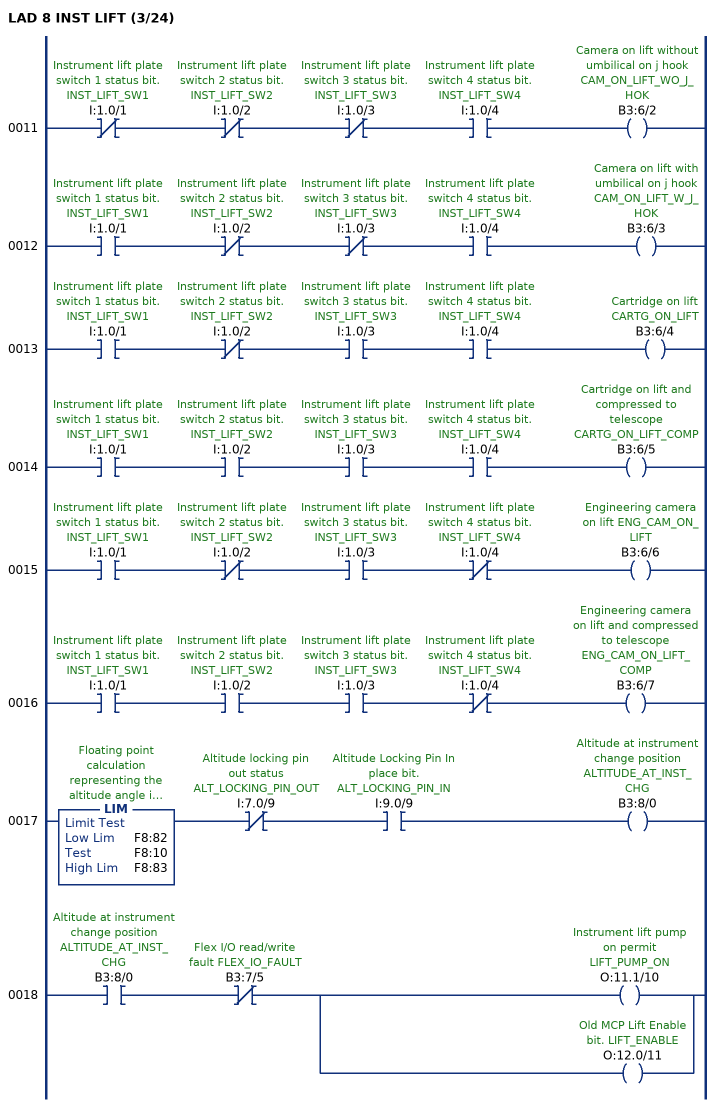
% Rung: 11 %
SOR XIO I:1.0/1 XIO I:1.0/2 XIO I:1.0/3 XIC I:1.0/4 OTE B3:6/2 EOR
%   I:1.0/1  INST_LIFT_SW1  "Instrument lift plate switch 1 status bit." %
%   I:1.0/2  INST_LIFT_SW2  "Instrument lift plate switch 2 status bit." %
%   I:1.0/3  INST_LIFT_SW3  "Instrument lift plate switch 3 status bit." %
%   I:1.0/4  INST_LIFT_SW4  "Instrument lift plate switch 4 status bit." %
%   B3:6/2  CAM_ON_LIFT_WO_J_HOK  "Camera on lift without umbilical on j hook" %
% Rung: 12 %
SOR XIC I:1.0/1 XIO I:1.0/2 XIO I:1.0/3 XIC I:1.0/4 OTE B3:6/3 EOR
%   I:1.0/1  INST_LIFT_SW1  "Instrument lift plate switch 1 status bit." %
%   I:1.0/2  INST_LIFT_SW2  "Instrument lift plate switch 2 status bit." %
%   I:1.0/3  INST_LIFT_SW3  "Instrument lift plate switch 3 status bit." %
%   I:1.0/4  INST_LIFT_SW4  "Instrument lift plate switch 4 status bit." %
%   B3:6/3  CAM_ON_LIFT_W_J_HOK  "Camera on lift with umbilical on j hook" %
% Rung: 13 %
SOR XIC I:1.0/1 XIO I:1.0/2 XIC I:1.0/3 XIC I:1.0/4 OTE B3:6/4 EOR
%   I:1.0/1  INST_LIFT_SW1  "Instrument lift plate switch 1 status bit." %
%   I:1.0/2  INST_LIFT_SW2  "Instrument lift plate switch 2 status bit." %
%   I:1.0/3  INST_LIFT_SW3  "Instrument lift plate switch 3 status bit." %
%   I:1.0/4  INST_LIFT_SW4  "Instrument lift plate switch 4 status bit." %
%   B3:6/4  CARTG_ON_LIFT  "Cartridge on lift" %
% Rung: 14 %
SOR XIC I:1.0/1 XIC I:1.0/2 XIC I:1.0/3 XIC I:1.0/4 OTE B3:6/5 EOR
%   I:1.0/1  INST_LIFT_SW1  "Instrument lift plate switch 1 status bit." %
%   I:1.0/2  INST_LIFT_SW2  "Instrument lift plate switch 2 status bit." %
%   I:1.0/3  INST_LIFT_SW3  "Instrument lift plate switch 3 status bit." %
%   I:1.0/4  INST_LIFT_SW4  "Instrument lift plate switch 4 status bit." %
%   B3:6/5  CARTG_ON_LIFT_COMP  "Cartridge on lift and compressed to telescope" %
% Rung: 15 %
SOR XIC I:1.0/1 XIO I:1.0/2 XIC I:1.0/3 XIO I:1.0/4 OTE B3:6/6 EOR
%   I:1.0/1  INST_LIFT_SW1  "Instrument lift plate switch 1 status bit." %
%   I:1.0/2  INST_LIFT_SW2  "Instrument lift plate switch 2 status bit." %
%   I:1.0/3  INST_LIFT_SW3  "Instrument lift plate switch 3 status bit." %
%   I:1.0/4  INST_LIFT_SW4  "Instrument lift plate switch 4 status bit." %
%   B3:6/6  ENG_CAM_ON_LIFT  "Engineering camera on lift" %
% Rung: 16 %
SOR XIC I:1.0/1 XIC I:1.0/2 XIC I:1.0/3 XIO I:1.0/4 OTE B3:6/7 EOR
%   I:1.0/1  INST_LIFT_SW1  "Instrument lift plate switch 1 status bit." %
%   I:1.0/2  INST_LIFT_SW2  "Instrument lift plate switch 2 status bit." %
%   I:1.0/3  INST_LIFT_SW3  "Instrument lift plate switch 3 status bit." %
%   I:1.0/4  INST_LIFT_SW4  "Instrument lift plate switch 4 status bit." %
%   B3:6/7  ENG_CAM_ON_LIFT_COMP  "Engineering camera on lift and compressed to telescope" %
% Rung: 17 %
SOR LIM F8:82 F8:10 F8:83 XIO I:7.0/9 XIC I:9.0/9 OTE B3:8/0 EOR
%   F8:82  INST_LIFT_LOW_LMT %
%   F8:10  ALT_ANGLE  "Floating point calculation representing the altitude angle in degrees." %
%   F8:83  INST_LIFT_HIGH_LMT %
%   I:7.0/9  ALT_LOCKING_PIN_OUT  "Altitude locking pin out status" %
%   I:9.0/9  ALT_LOCKING_PIN_IN  "Altitude Locking Pin In place bit." %
%   B3:8/0  ALTITUDE_AT_INST_CHG  "Altitude at instrument change position" %
% Rung: 18 %
SOR XIC B3:8/0 XIO B3:7/5 BST OTE O:11.1/10 NXB OTE O:12.0/11 BND EOR
%   B3:8/0  ALTITUDE_AT_INST_CHG  "Altitude at instrument change position" %
%   B3:7/5  FLEX_IO_FAULT  "Flex I/O read/write fault" %
%   O:11.1/10  LIFT_PUMP_ON  "Instrument lift pump on permit" %
%   O:12.0/11  LIFT_ENABLE  "Old MCP Lift Enable bit." %

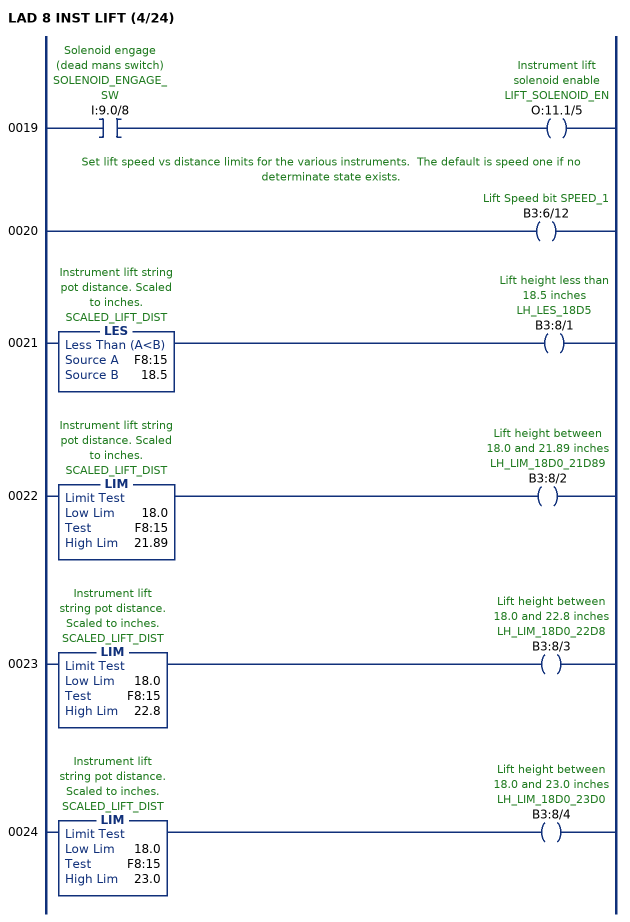
% Rung: 19 %
SOR XIC I:9.0/8 OTE O:11.1/5 EOR
%   I:9.0/8  SOLENOID_ENGAGE_SW  "Solenoid engage (dead mans switch)" %
%   O:11.1/5  LIFT_SOLENOID_EN  "Instrument lift solenoid enable" %
% Rung: 20 %
% Set lift speed vs distance limits for the various instruments.  The default is speed one if no determinate state exists. %
SOR OTE B3:6/12 EOR
%   B3:6/12  SPEED_1  "Lift Speed bit" %
% Rung: 21 %
SOR LES F8:15 18.5 OTE B3:8/1 EOR
%   F8:15  SCALED_LIFT_DIST  "Instrument lift string pot distance. Scaled to inches." %
%   B3:8/1  LH_LES_18D5  "Lift height less than 18.5 inches" %
% Rung: 22 %
SOR LIM 18.0 F8:15 21.89 OTE B3:8/2 EOR
%   F8:15  SCALED_LIFT_DIST  "Instrument lift string pot distance. Scaled to inches." %
%   B3:8/2  LH_LIM_18D0_21D89  "Lift height between 18.0 and 21.89 inches" %
% Rung: 23 %
SOR LIM 18.0 F8:15 22.8 OTE B3:8/3 EOR
%   F8:15  SCALED_LIFT_DIST  "Instrument lift string pot distance. Scaled to inches." %
%   B3:8/3  LH_LIM_18D0_22D8  "Lift height between 18.0 and 22.8 inches" %
% Rung: 24 %
SOR LIM 18.0 F8:15 23.0 OTE B3:8/4 EOR
%   F8:15  SCALED_LIFT_DIST  "Instrument lift string pot distance. Scaled to inches." %
%   B3:8/4  LH_LIM_18D0_23D0  "Lift height between 18.0 and 23.0 inches" %

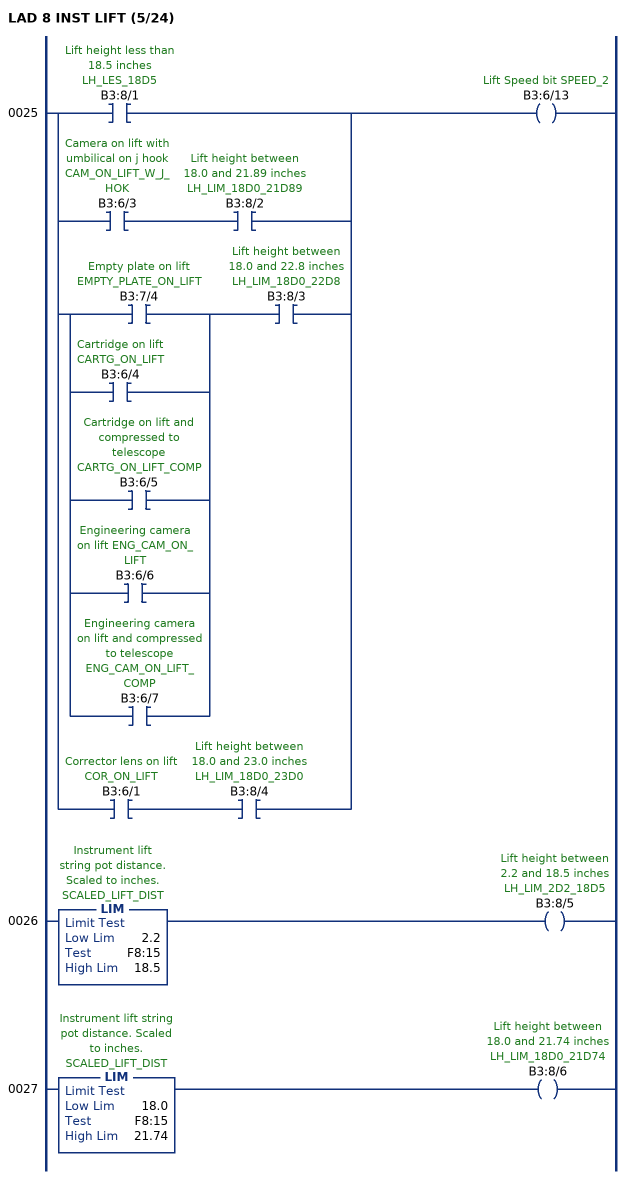
% Rung: 25 %
SOR BST XIC B3:8/1 NXB XIC B3:6/3 XIC B3:8/2 NXB BST XIC B3:7/4 NXB XIC B3:6/4 NXB XIC B3:6/5 NXB XIC B3:6/6 NXB XIC B3:6/7 BND XIC B3:8/3 NXB XIC B3:6/1 XIC B3:8/4 BND OTE B3:6/13 EOR
%   B3:8/1  LH_LES_18D5  "Lift height less than 18.5 inches" %
%   B3:6/3  CAM_ON_LIFT_W_J_HOK  "Camera on lift with umbilical on j hook" %
%   B3:8/2  LH_LIM_18D0_21D89  "Lift height between 18.0 and 21.89 inches" %
%   B3:7/4  EMPTY_PLATE_ON_LIFT  "Empty plate on lift" %
%   B3:6/4  CARTG_ON_LIFT  "Cartridge on lift" %
%   B3:6/5  CARTG_ON_LIFT_COMP  "Cartridge on lift and compressed to telescope" %
%   B3:6/6  ENG_CAM_ON_LIFT  "Engineering camera on lift" %
%   B3:6/7  ENG_CAM_ON_LIFT_COMP  "Engineering camera on lift and compressed to telescope" %
%   B3:8/3  LH_LIM_18D0_22D8  "Lift height between 18.0 and 22.8 inches" %
%   B3:6/1  COR_ON_LIFT  "Corrector lens on lift" %
%   B3:8/4  LH_LIM_18D0_23D0  "Lift height between 18.0 and 23.0 inches" %
%   B3:6/13  SPEED_2  "Lift Speed bit" %
% Rung: 26 %
SOR LIM 2.2 F8:15 18.5 OTE B3:8/5 EOR
%   F8:15  SCALED_LIFT_DIST  "Instrument lift string pot distance. Scaled to inches." %
%   B3:8/5  LH_LIM_2D2_18D5  "Lift height between 2.2 and 18.5 inches" %
% Rung: 27 %
SOR LIM 18.0 F8:15 21.74 OTE B3:8/6 EOR
%   F8:15  SCALED_LIFT_DIST  "Instrument lift string pot distance. Scaled to inches." %
%   B3:8/6  LH_LIM_18D0_21D74  "Lift height between 18.0 and 21.74 inches" %

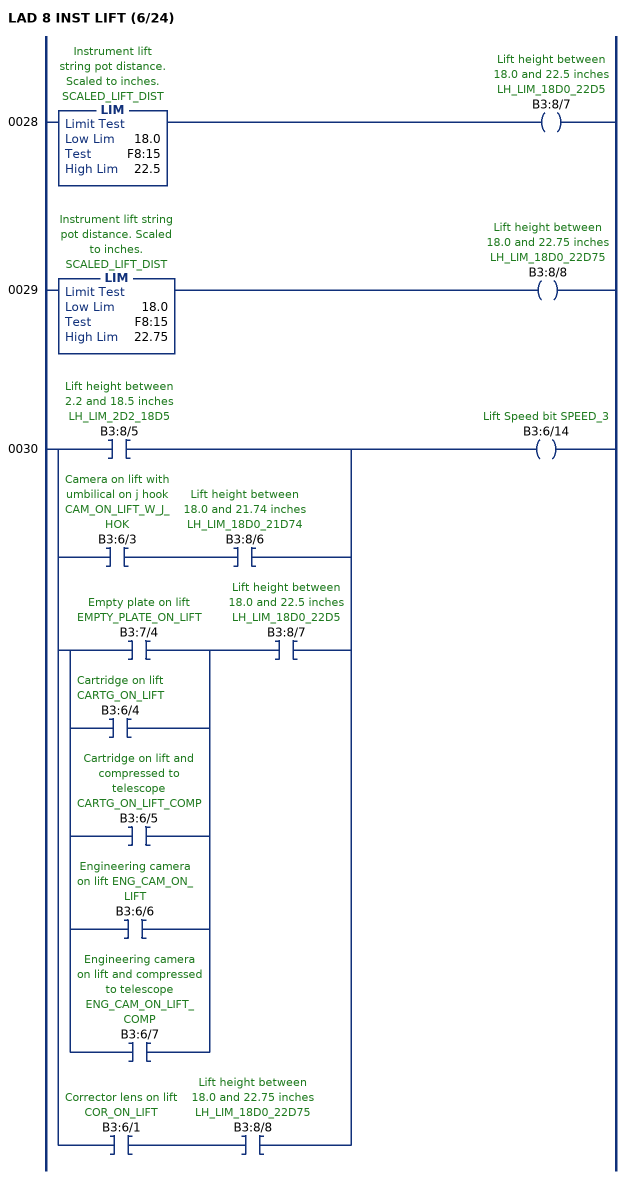
% Rung: 28 %
SOR LIM 18.0 F8:15 22.5 OTE B3:8/7 EOR
%   F8:15  SCALED_LIFT_DIST  "Instrument lift string pot distance. Scaled to inches." %
%   B3:8/7  LH_LIM_18D0_22D5  "Lift height between 18.0 and 22.5 inches" %
% Rung: 29 %
SOR LIM 18.0 F8:15 22.75 OTE B3:8/8 EOR
%   F8:15  SCALED_LIFT_DIST  "Instrument lift string pot distance. Scaled to inches." %
%   B3:8/8  LH_LIM_18D0_22D75  "Lift height between 18.0 and 22.75 inches" %
% Rung: 30 %
SOR BST XIC B3:8/5 NXB XIC B3:6/3 XIC B3:8/6 NXB BST XIC B3:7/4 NXB XIC B3:6/4 NXB XIC B3:6/5 NXB XIC B3:6/6 NXB XIC B3:6/7 BND XIC B3:8/7 NXB XIC B3:6/1 XIC B3:8/8 BND OTE B3:6/14 EOR
%   B3:8/5  LH_LIM_2D2_18D5  "Lift height between 2.2 and 18.5 inches" %
%   B3:6/3  CAM_ON_LIFT_W_J_HOK  "Camera on lift with umbilical on j hook" %
%   B3:8/6  LH_LIM_18D0_21D74  "Lift height between 18.0 and 21.74 inches" %
%   B3:7/4  EMPTY_PLATE_ON_LIFT  "Empty plate on lift" %
%   B3:6/4  CARTG_ON_LIFT  "Cartridge on lift" %
%   B3:6/5  CARTG_ON_LIFT_COMP  "Cartridge on lift and compressed to telescope" %
%   B3:6/6  ENG_CAM_ON_LIFT  "Engineering camera on lift" %
%   B3:6/7  ENG_CAM_ON_LIFT_COMP  "Engineering camera on lift and compressed to telescope" %
%   B3:8/7  LH_LIM_18D0_22D5  "Lift height between 18.0 and 22.5 inches" %
%   B3:6/1  COR_ON_LIFT  "Corrector lens on lift" %
%   B3:8/8  LH_LIM_18D0_22D75  "Lift height between 18.0 and 22.75 inches" %
%   B3:6/14  SPEED_3  "Lift Speed bit" %

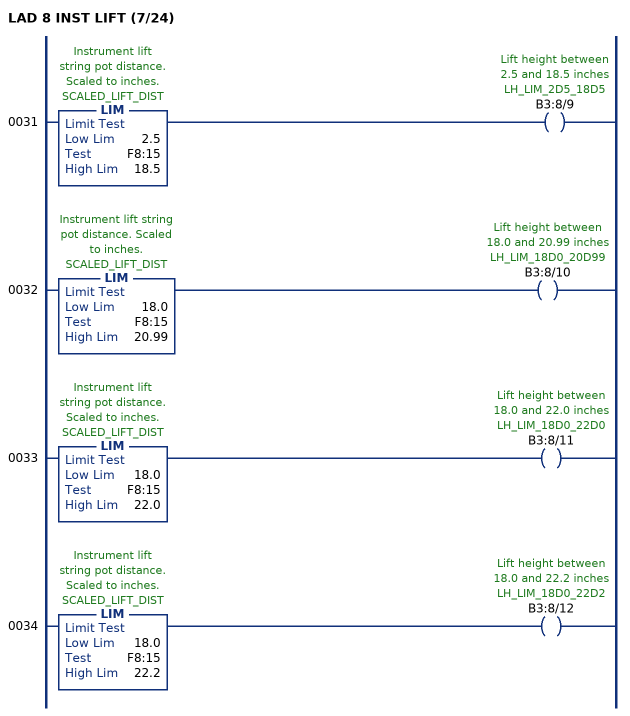
% Rung: 31 %
SOR LIM 2.5 F8:15 18.5 OTE B3:8/9 EOR
%   F8:15  SCALED_LIFT_DIST  "Instrument lift string pot distance. Scaled to inches." %
%   B3:8/9  LH_LIM_2D5_18D5  "Lift height between 2.5 and 18.5 inches" %
% Rung: 32 %
SOR LIM 18.0 F8:15 20.99 OTE B3:8/10 EOR
%   F8:15  SCALED_LIFT_DIST  "Instrument lift string pot distance. Scaled to inches." %
%   B3:8/10  LH_LIM_18D0_20D99  "Lift height between 18.0 and 20.99 inches" %
% Rung: 33 %
SOR LIM 18.0 F8:15 22.0 OTE B3:8/11 EOR
%   F8:15  SCALED_LIFT_DIST  "Instrument lift string pot distance. Scaled to inches." %
%   B3:8/11  LH_LIM_18D0_22D0  "Lift height between 18.0 and 22.0 inches" %
% Rung: 34 %
SOR LIM 18.0 F8:15 22.2 OTE B3:8/12 EOR
%   F8:15  SCALED_LIFT_DIST  "Instrument lift string pot distance. Scaled to inches." %
%   B3:8/12  LH_LIM_18D0_22D2  "Lift height between 18.0 and 22.2 inches" %

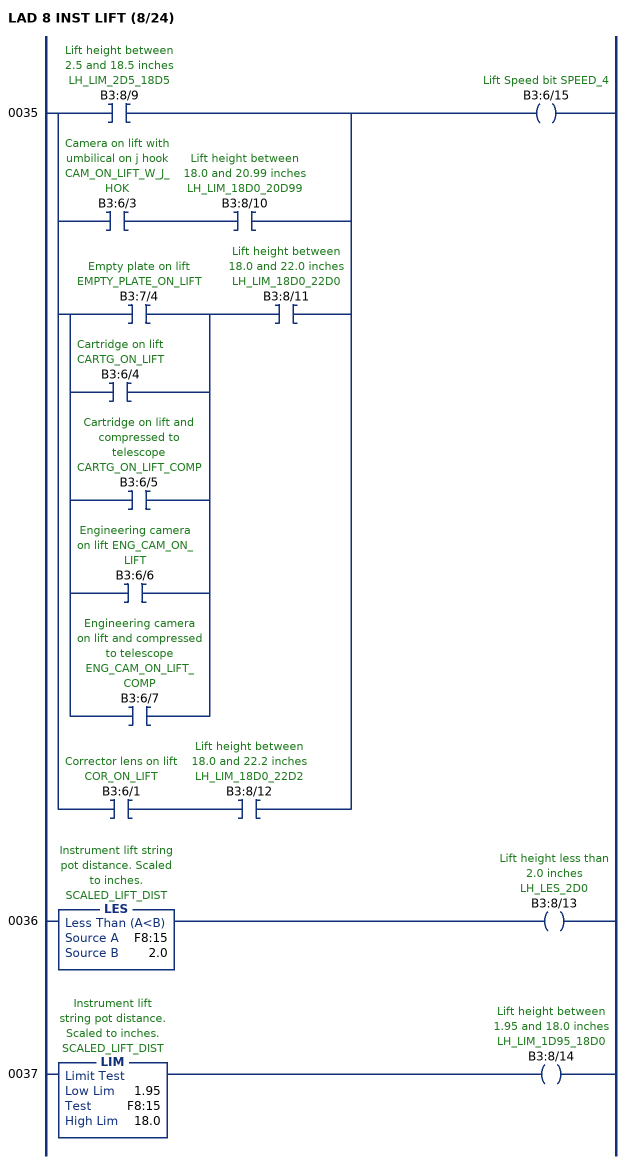
% Rung: 35 %
SOR BST XIC B3:8/9 NXB XIC B3:6/3 XIC B3:8/10 NXB BST XIC B3:7/4 NXB XIC B3:6/4 NXB XIC B3:6/5 NXB XIC B3:6/6 NXB XIC B3:6/7 BND XIC B3:8/11 NXB XIC B3:6/1 XIC B3:8/12 BND OTE B3:6/15 EOR
%   B3:8/9  LH_LIM_2D5_18D5  "Lift height between 2.5 and 18.5 inches" %
%   B3:6/3  CAM_ON_LIFT_W_J_HOK  "Camera on lift with umbilical on j hook" %
%   B3:8/10  LH_LIM_18D0_20D99  "Lift height between 18.0 and 20.99 inches" %
%   B3:7/4  EMPTY_PLATE_ON_LIFT  "Empty plate on lift" %
%   B3:6/4  CARTG_ON_LIFT  "Cartridge on lift" %
%   B3:6/5  CARTG_ON_LIFT_COMP  "Cartridge on lift and compressed to telescope" %
%   B3:6/6  ENG_CAM_ON_LIFT  "Engineering camera on lift" %
%   B3:6/7  ENG_CAM_ON_LIFT_COMP  "Engineering camera on lift and compressed to telescope" %
%   B3:8/11  LH_LIM_18D0_22D0  "Lift height between 18.0 and 22.0 inches" %
%   B3:6/1  COR_ON_LIFT  "Corrector lens on lift" %
%   B3:8/12  LH_LIM_18D0_22D2  "Lift height between 18.0 and 22.2 inches" %
%   B3:6/15  SPEED_4  "Lift Speed bit" %
% Rung: 36 %
SOR LES F8:15 2.0 OTE B3:8/13 EOR
%   F8:15  SCALED_LIFT_DIST  "Instrument lift string pot distance. Scaled to inches." %
%   B3:8/13  LH_LES_2D0  "Lift height less than 2.0 inches" %
% Rung: 37 %
SOR LIM 1.95 F8:15 18.0 OTE B3:8/14 EOR
%   F8:15  SCALED_LIFT_DIST  "Instrument lift string pot distance. Scaled to inches." %
%   B3:8/14  LH_LIM_1D95_18D0  "Lift height between 1.95 and 18.0 inches" %

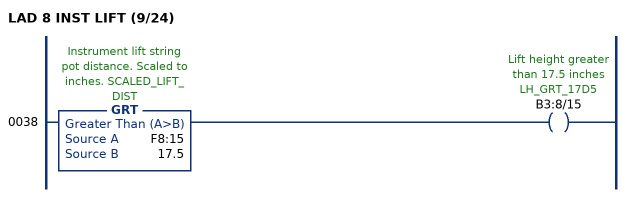
% Rung: 38 %
SOR GRT F8:15 17.5 OTE B3:8/15 EOR
%   F8:15  SCALED_LIFT_DIST  "Instrument lift string pot distance. Scaled to inches." %
%   B3:8/15  LH_GRT_17D5  "Lift height greater than 17.5 inches" %

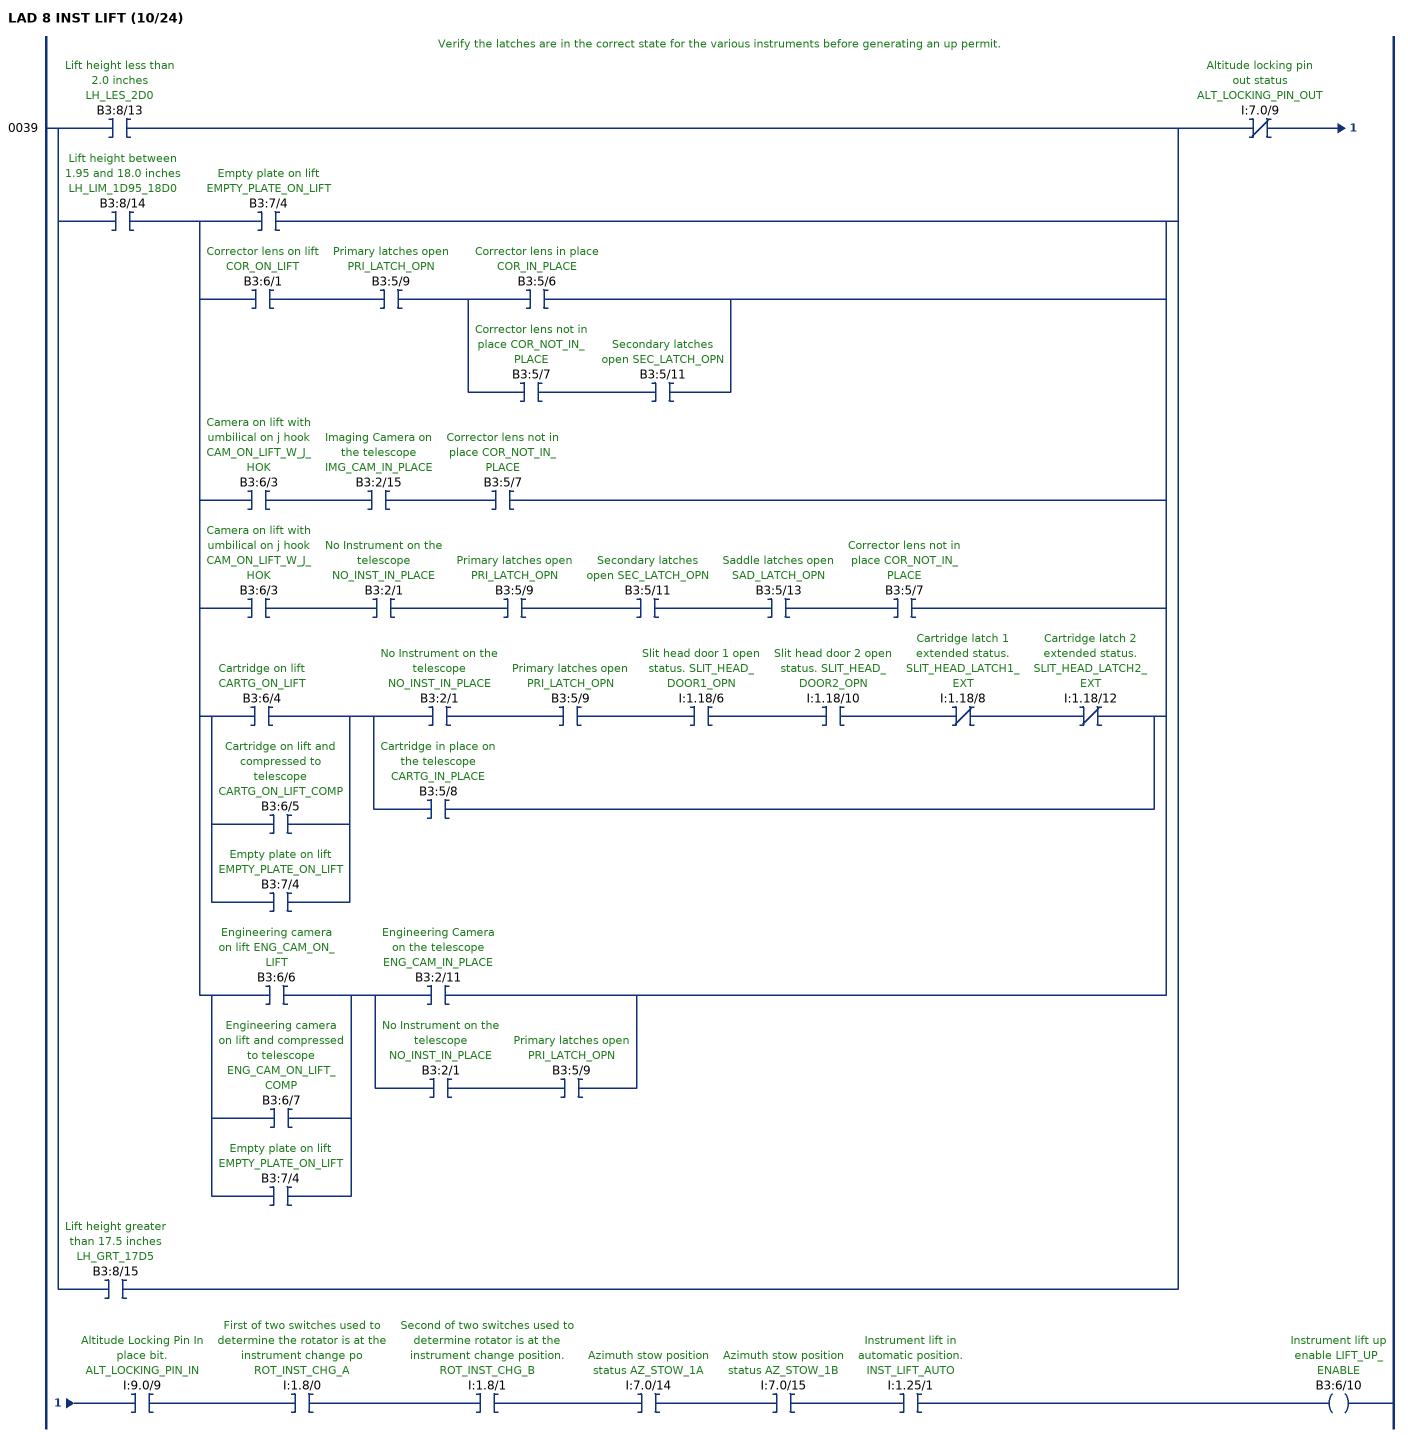
% Rung: 39 %
% Verify the latches are in the correct state for the various instruments before generating an up permit. %
SOR BST XIC B3:8/13 NXB XIC B3:8/14 BST XIC B3:7/4 NXB XIC B3:6/1 XIC B3:5/9 BST XIC B3:5/6 NXB XIC B3:5/7 XIC B3:5/11 BND NXB BST XIC B3:6/3 XIC B3:2/15 XIC B3:5/7 NXB XIC B3:6/3 XIC B3:2/1 XIC B3:5/9 XIC B3:5/11 XIC B3:5/13 XIC B3:5/7 BND NXB BST XIC B3:6/4 NXB XIC B3:6/5 NXB XIC B3:7/4 BND BST XIC B3:2/1 XIC B3:5/9 XIC I:1.18/6 XIC I:1.18/10 XIO I:1.18/8 XIO I:1.18/12 NXB XIC B3:5/8 BND NXB BST XIC B3:6/6 NXB XIC B3:6/7 NXB XIC B3:7/4 BND BST XIC B3:2/11 NXB XIC B3:2/1 XIC B3:5/9 BND BND NXB XIC B3:8/15 BND XIO I:7.0/9 XIC I:9.0/9 XIC I:1.8/0 XIC I:1.8/1 XIC I:7.0/14 XIC I:7.0/15 XIC I:1.25/1 OTE B3:6/10 EOR
%   B3:8/13  LH_LES_2D0  "Lift height less than 2.0 inches" %
%   B3:8/14  LH_LIM_1D95_18D0  "Lift height between 1.95 and 18.0 inches" %
%   B3:7/4  EMPTY_PLATE_ON_LIFT  "Empty plate on lift" %
%   B3:6/1  COR_ON_LIFT  "Corrector lens on lift" %
%   B3:5/9  PRI_LATCH_OPN  "Primary latches open" %
%   B3:5/6  COR_IN_PLACE  "Corrector lens in place" %
%   B3:5/7  COR_NOT_IN_PLACE  "Corrector lens not in place" %
%   B3:5/11  SEC_LATCH_OPN  "Secondary latches open" %
%   B3:6/3  CAM_ON_LIFT_W_J_HOK  "Camera on lift with umbilical on j hook" %
%   B3:2/15  IMG_CAM_IN_PLACE  "Imaging Camera on the telescope" %
%   B3:2/1  NO_INST_IN_PLACE  "No Instrument on the telescope" %
%   B3:5/13  SAD_LATCH_OPN  "Saddle latches open" %
%   B3:6/4  CARTG_ON_LIFT  "Cartridge on lift" %
%   B3:6/5  CARTG_ON_LIFT_COMP  "Cartridge on lift and compressed to telescope" %
%   I:1.18/6  SLIT_HEAD_DOOR1_OPN  "Slit head door 1 open status." %
%   I:1.18/10  SLIT_HEAD_DOOR2_OPN  "Slit head door 2 open status." %
%   I:1.18/8  SLIT_HEAD_LATCH1_EXT  "Cartridge latch 1 extended status." %
%   I:1.18/12  SLIT_HEAD_LATCH2_EXT  "Cartridge latch 2 extended status." %
%   B3:5/8  CARTG_IN_PLACE  "Cartridge in place on the telescope" %
%   B3:6/6  ENG_CAM_ON_LIFT  "Engineering camera on lift" %
%   B3:6/7  ENG_CAM_ON_LIFT_COMP  "Engineering camera on lift and compressed to telescope" %
%   B3:2/11  ENG_CAM_IN_PLACE  "Engineering Camera on the telescope" %
%   B3:8/15  LH_GRT_17D5  "Lift height greater than 17.5 inches" %
%   I:7.0/9  ALT_LOCKING_PIN_OUT  "Altitude locking pin out status" %
%   I:9.0/9  ALT_LOCKING_PIN_IN  "Altitude Locking Pin In place bit." %
%   I:1.8/0  ROT_INST_CHG_A  "First of two switches used to determine the rotator is at the instrument change po" %
%   I:1.8/1  ROT_INST_CHG_B  "Second of two switches used to determine rotator is at the instrument change position." %
%   I:7.0/14  AZ_STOW_1A  "Azimuth stow position status" %
%   I:7.0/15  AZ_STOW_1B  "Azimuth stow position status" %
%   I:1.25/1  INST_LIFT_AUTO  "Instrument lift in automatic position." %
%   B3:6/10  LIFT_UP_ENABLE  "Instrument lift up enable" %

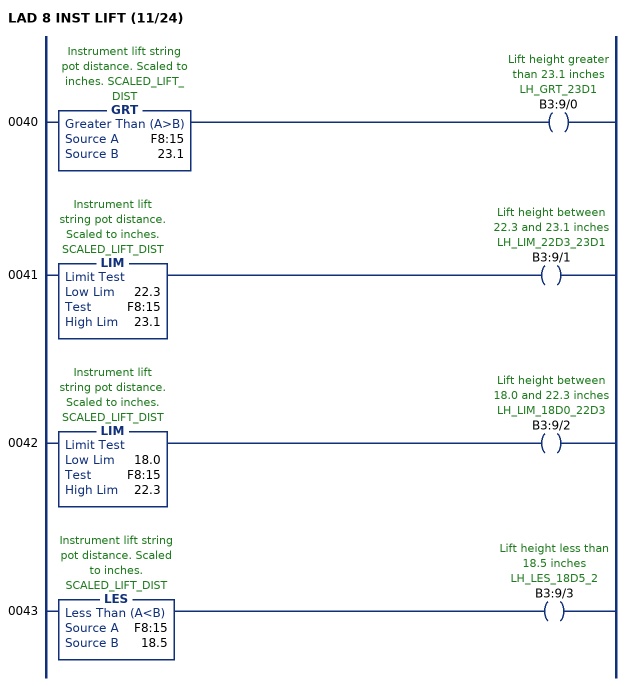
% Rung: 40 %
SOR GRT F8:15 23.1 OTE B3:9/0 EOR
%   F8:15  SCALED_LIFT_DIST  "Instrument lift string pot distance. Scaled to inches." %
%   B3:9/0  LH_GRT_23D1  "Lift height greater than 23.1 inches" %
% Rung: 41 %
SOR LIM 22.3 F8:15 23.1 OTE B3:9/1 EOR
%   F8:15  SCALED_LIFT_DIST  "Instrument lift string pot distance. Scaled to inches." %
%   B3:9/1  LH_LIM_22D3_23D1  "Lift height between 22.3 and 23.1 inches" %
% Rung: 42 %
SOR LIM 18.0 F8:15 22.3 OTE B3:9/2 EOR
%   F8:15  SCALED_LIFT_DIST  "Instrument lift string pot distance. Scaled to inches." %
%   B3:9/2  LH_LIM_18D0_22D3  "Lift height between 18.0 and 22.3 inches" %
% Rung: 43 %
SOR LES F8:15 18.5 OTE B3:9/3 EOR
%   F8:15  SCALED_LIFT_DIST  "Instrument lift string pot distance. Scaled to inches." %
%   B3:9/3  LH_LES_18D5_2  "Lift height less than 18.5 inches" %

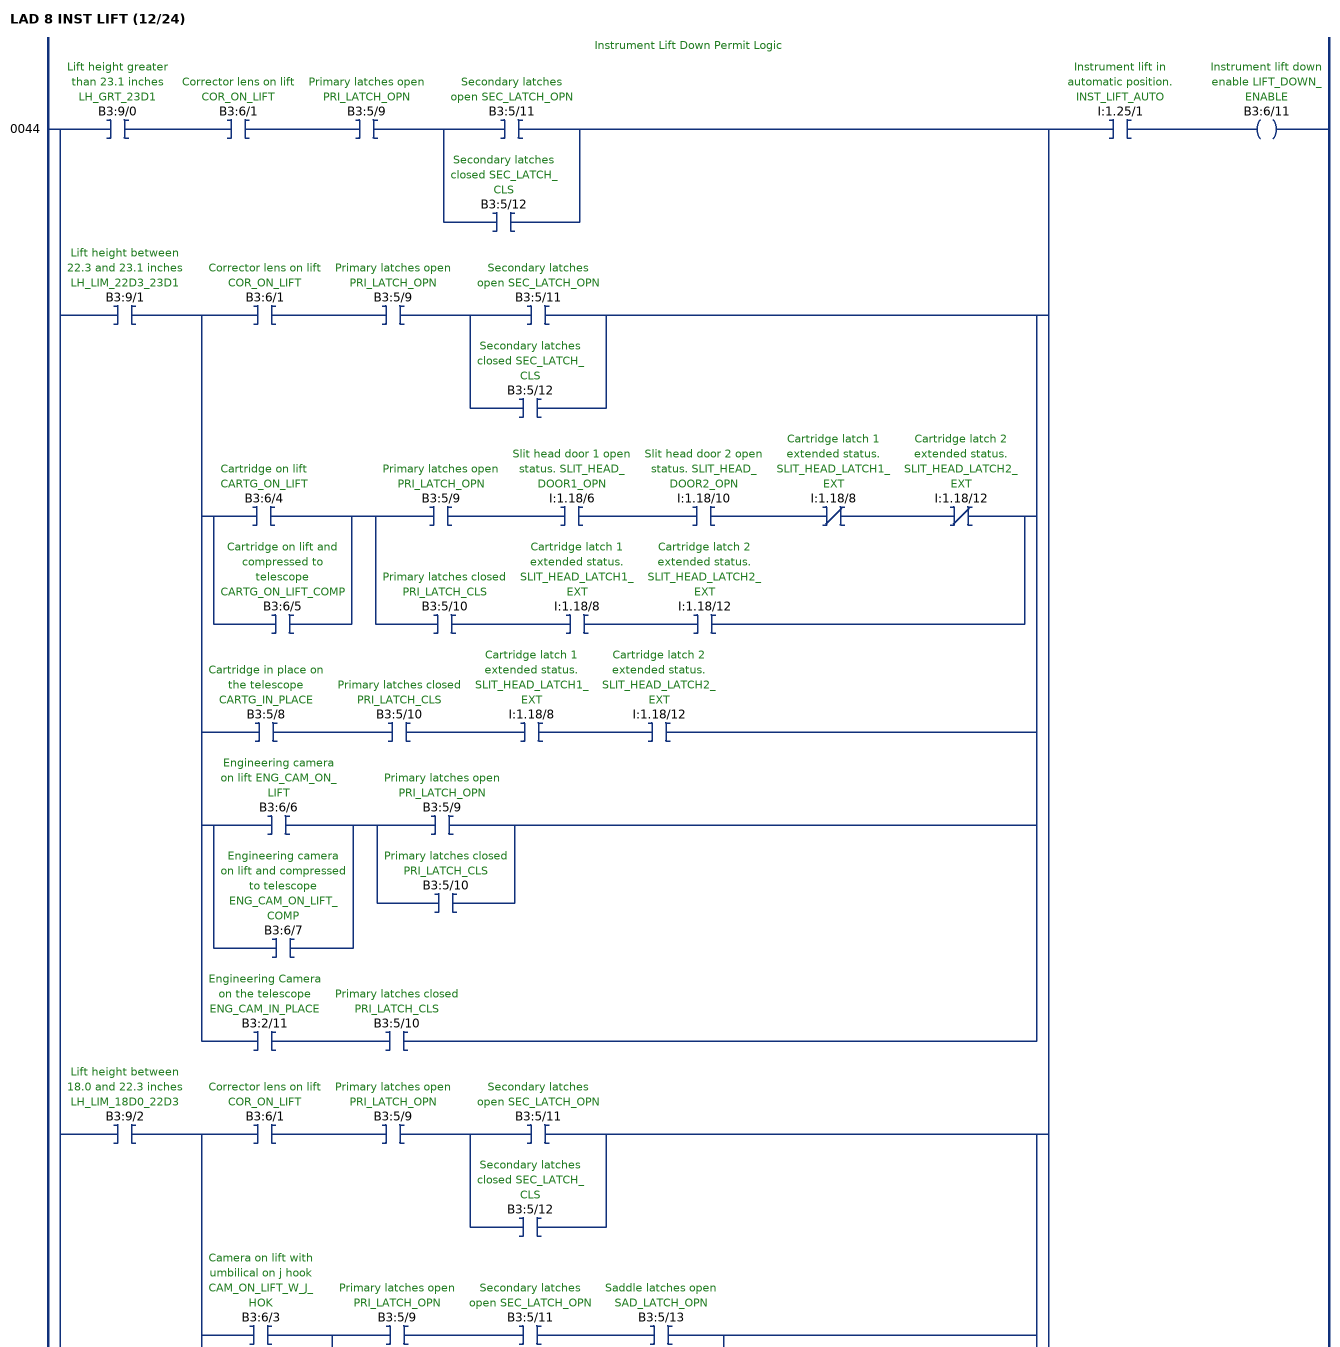

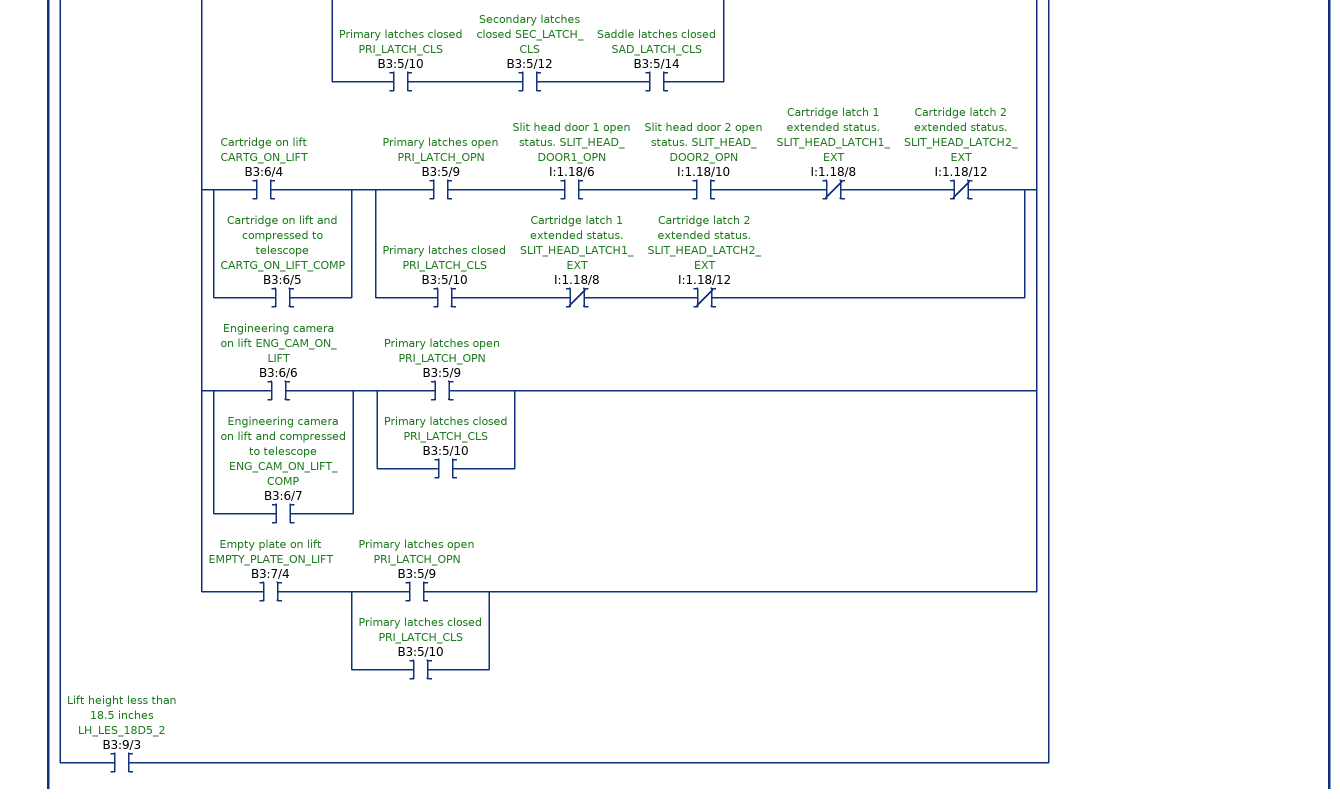
% Rung: 44 %
% Instrument Lift Down Permit Logic %
SOR BST XIC B3:9/0 XIC B3:6/1 XIC B3:5/9 BST XIC B3:5/11 NXB XIC B3:5/12 BND NXB XIC B3:9/1 BST XIC B3:6/1 XIC B3:5/9 BST XIC B3:5/11 NXB XIC B3:5/12 BND NXB BST XIC B3:6/4 NXB XIC B3:6/5 BND BST XIC B3:5/9 XIC I:1.18/6 XIC I:1.18/10 XIO I:1.18/8 XIO I:1.18/12 NXB XIC B3:5/10 XIC I:1.18/8 XIC I:1.18/12 BND NXB XIC B3:5/8 XIC B3:5/10 XIC I:1.18/8 XIC I:1.18/12 NXB BST XIC B3:6/6 NXB XIC B3:6/7 BND BST XIC B3:5/9 NXB XIC B3:5/10 BND NXB XIC B3:2/11 XIC B3:5/10 BND NXB XIC B3:9/2 BST XIC B3:6/1 XIC B3:5/9 BST XIC B3:5/11 NXB XIC B3:5/12 BND NXB XIC B3:6/3 BST XIC B3:5/9 XIC B3:5/11 XIC B3:5/13 NXB XIC B3:5/10 XIC B3:5/12 XIC B3:5/14 BND NXB BST XIC B3:6/4 NXB XIC B3:6/5 BND BST XIC B3:5/9 XIC I:1.18/6 XIC I:1.18/10 XIO I:1.18/8 XIO I:1.18/12 NXB XIC B3:5/10 XIO I:1.18/8 XIO I:1.18/12 BND NXB BST XIC B3:6/6 NXB XIC B3:6/7 BND BST XIC B3:5/9 NXB XIC B3:5/10 BND NXB XIC B3:7/4 BST XIC B3:5/9 NXB XIC B3:5/10 BND BND NXB XIC B3:9/3 BND XIC I:1.25/1 OTE B3:6/11 EOR
%   B3:9/0  LH_GRT_23D1  "Lift height greater than 23.1 inches" %
%   B3:6/1  COR_ON_LIFT  "Corrector lens on lift" %
%   B3:5/9  PRI_LATCH_OPN  "Primary latches open" %
%   B3:5/11  SEC_LATCH_OPN  "Secondary latches open" %
%   B3:5/12  SEC_LATCH_CLS  "Secondary latches closed" %
%   B3:9/1  LH_LIM_22D3_23D1  "Lift height between 22.3 and 23.1 inches" %
%   B3:6/4  CARTG_ON_LIFT  "Cartridge on lift" %
%   B3:6/5  CARTG_ON_LIFT_COMP  "Cartridge on lift and compressed to telescope" %
%   I:1.18/6  SLIT_HEAD_DOOR1_OPN  "Slit head door 1 open status." %
%   I:1.18/10  SLIT_HEAD_DOOR2_OPN  "Slit head door 2 open status." %
%   I:1.18/8  SLIT_HEAD_LATCH1_EXT  "Cartridge latch 1 extended status." %
%   I:1.18/12  SLIT_HEAD_LATCH2_EXT  "Cartridge latch 2 extended status." %
%   B3:5/10  PRI_LATCH_CLS  "Primary latches closed" %
%   B3:5/8  CARTG_IN_PLACE  "Cartridge in place on the telescope" %
%   B3:6/6  ENG_CAM_ON_LIFT  "Engineering camera on lift" %
%   B3:6/7  ENG_CAM_ON_LIFT_COMP  "Engineering camera on lift and compressed to telescope" %
%   B3:2/11  ENG_CAM_IN_PLACE  "Engineering Camera on the telescope" %
%   B3:9/2  LH_LIM_18D0_22D3  "Lift height between 18.0 and 22.3 inches" %
%   B3:6/3  CAM_ON_LIFT_W_J_HOK  "Camera on lift with umbilical on j hook" %
%   B3:5/13  SAD_LATCH_OPN  "Saddle latches open" %
%   B3:5/14  SAD_LATCH_CLS  "Saddle latches closed" %
%   B3:7/4  EMPTY_PLATE_ON_LIFT  "Empty plate on lift" %
%   B3:9/3  LH_LES_18D5_2  "Lift height less than 18.5 inches" %
%   I:1.25/1  INST_LIFT_AUTO  "Instrument lift in automatic position." %
%   B3:6/11  LIFT_DOWN_ENABLE  "Instrument lift down enable" %

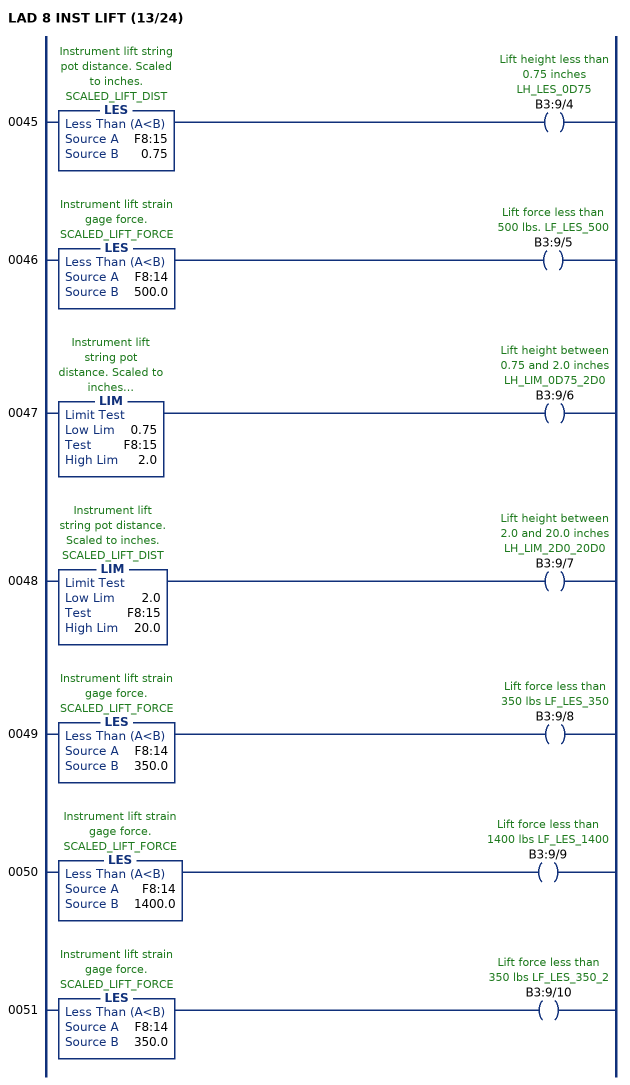
% Rung: 45 %
SOR LES F8:15 0.75 OTE B3:9/4 EOR
%   F8:15  SCALED_LIFT_DIST  "Instrument lift string pot distance. Scaled to inches." %
%   B3:9/4  LH_LES_0D75  "Lift height less than 0.75 inches" %
% Rung: 46 %
SOR LES F8:14 500.0 OTE B3:9/5 EOR
%   F8:14  SCALED_LIFT_FORCE  "Instrument lift strain gage force." %
%   B3:9/5  LF_LES_500  "Lift force less than 500 lbs." %
% Rung: 47 %
SOR LIM 0.75 F8:15 2.0 OTE B3:9/6 EOR
%   F8:15  SCALED_LIFT_DIST  "Instrument lift string pot distance. Scaled to inches." %
%   B3:9/6  LH_LIM_0D75_2D0  "Lift height between 0.75 and 2.0 inches" %
% Rung: 48 %
SOR LIM 2.0 F8:15 20.0 OTE B3:9/7 EOR
%   F8:15  SCALED_LIFT_DIST  "Instrument lift string pot distance. Scaled to inches." %
%   B3:9/7  LH_LIM_2D0_20D0  "Lift height between 2.0 and 20.0 inches" %
% Rung: 49 %
SOR LES F8:14 350.0 OTE B3:9/8 EOR
%   F8:14  SCALED_LIFT_FORCE  "Instrument lift strain gage force." %
%   B3:9/8  LF_LES_350  "Lift force less than 350 lbs" %
% Rung: 50 %
SOR LES F8:14 1400.0 OTE B3:9/9 EOR
%   F8:14  SCALED_LIFT_FORCE  "Instrument lift strain gage force." %
%   B3:9/9  LF_LES_1400  "Lift force less than 1400 lbs" %
% Rung: 51 %
SOR LES F8:14 350.0 OTE B3:9/10 EOR
%   F8:14  SCALED_LIFT_FORCE  "Instrument lift strain gage force." %
%   B3:9/10  LF_LES_350_2  "Lift force less than 350 lbs" %

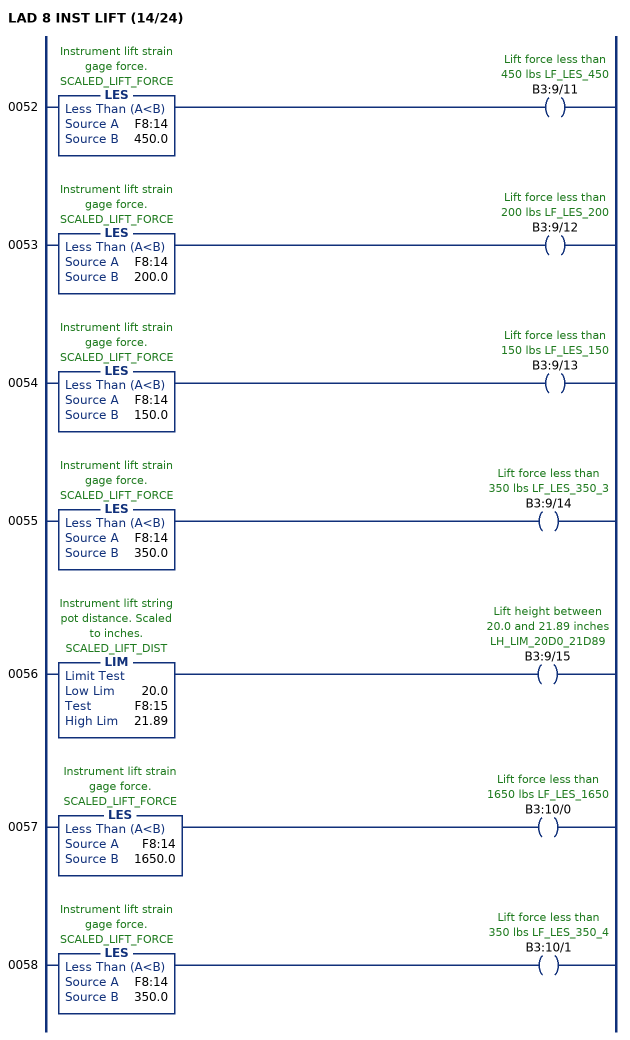
% Rung: 52 %
SOR LES F8:14 450.0 OTE B3:9/11 EOR
%   F8:14  SCALED_LIFT_FORCE  "Instrument lift strain gage force." %
%   B3:9/11  LF_LES_450  "Lift force less than 450 lbs" %
% Rung: 53 %
SOR LES F8:14 200.0 OTE B3:9/12 EOR
%   F8:14  SCALED_LIFT_FORCE  "Instrument lift strain gage force." %
%   B3:9/12  LF_LES_200  "Lift force less than 200 lbs" %
% Rung: 54 %
SOR LES F8:14 150.0 OTE B3:9/13 EOR
%   F8:14  SCALED_LIFT_FORCE  "Instrument lift strain gage force." %
%   B3:9/13  LF_LES_150  "Lift force less than 150 lbs" %
% Rung: 55 %
SOR LES F8:14 350.0 OTE B3:9/14 EOR
%   F8:14  SCALED_LIFT_FORCE  "Instrument lift strain gage force." %
%   B3:9/14  LF_LES_350_3  "Lift force less than 350 lbs" %
% Rung: 56 %
SOR LIM 20.0 F8:15 21.89 OTE B3:9/15 EOR
%   F8:15  SCALED_LIFT_DIST  "Instrument lift string pot distance. Scaled to inches." %
%   B3:9/15  LH_LIM_20D0_21D89  "Lift height between 20.0 and 21.89 inches" %
% Rung: 57 %
SOR LES F8:14 1650.0 OTE B3:10/0 EOR
%   F8:14  SCALED_LIFT_FORCE  "Instrument lift strain gage force." %
%   B3:10/0  LF_LES_1650  "Lift force less than 1650 lbs" %
% Rung: 58 %
SOR LES F8:14 350.0 OTE B3:10/1 EOR
%   F8:14  SCALED_LIFT_FORCE  "Instrument lift strain gage force." %
%   B3:10/1  LF_LES_350_4  "Lift force less than 350 lbs" %

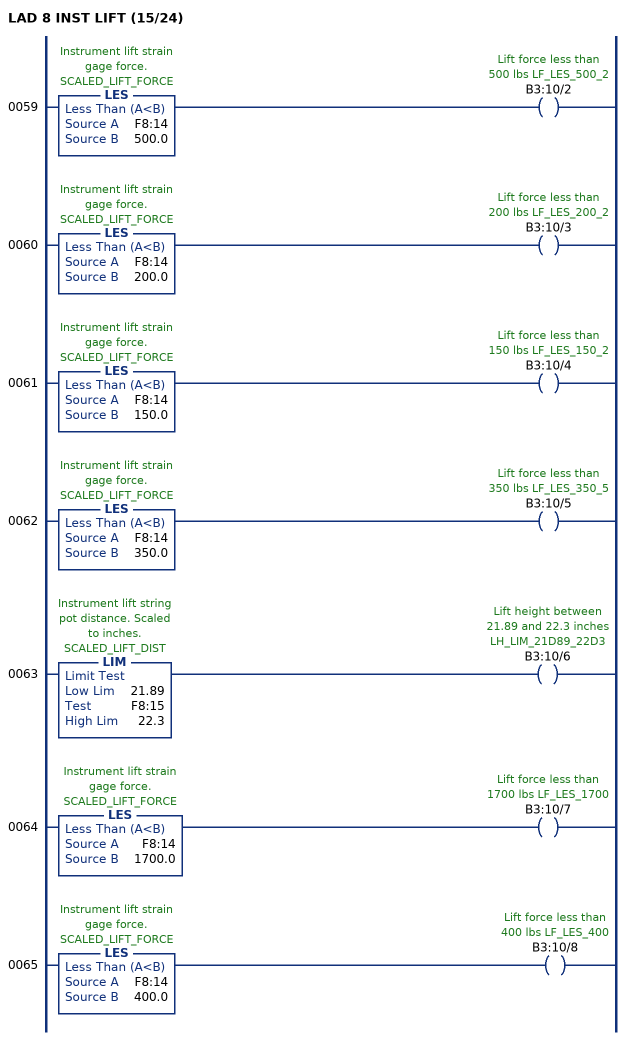
% Rung: 59 %
SOR LES F8:14 500.0 OTE B3:10/2 EOR
%   F8:14  SCALED_LIFT_FORCE  "Instrument lift strain gage force." %
%   B3:10/2  LF_LES_500_2  "Lift force less than 500 lbs" %
% Rung: 60 %
SOR LES F8:14 200.0 OTE B3:10/3 EOR
%   F8:14  SCALED_LIFT_FORCE  "Instrument lift strain gage force." %
%   B3:10/3  LF_LES_200_2  "Lift force less than 200 lbs" %
% Rung: 61 %
SOR LES F8:14 150.0 OTE B3:10/4 EOR
%   F8:14  SCALED_LIFT_FORCE  "Instrument lift strain gage force." %
%   B3:10/4  LF_LES_150_2  "Lift force less than 150 lbs" %
% Rung: 62 %
SOR LES F8:14 350.0 OTE B3:10/5 EOR
%   F8:14  SCALED_LIFT_FORCE  "Instrument lift strain gage force." %
%   B3:10/5  LF_LES_350_5  "Lift force less than 350 lbs" %
% Rung: 63 %
SOR LIM 21.89 F8:15 22.3 OTE B3:10/6 EOR
%   F8:15  SCALED_LIFT_DIST  "Instrument lift string pot distance. Scaled to inches." %
%   B3:10/6  LH_LIM_21D89_22D3  "Lift height between 21.89 and 22.3 inches" %
% Rung: 64 %
SOR LES F8:14 1700.0 OTE B3:10/7 EOR
%   F8:14  SCALED_LIFT_FORCE  "Instrument lift strain gage force." %
%   B3:10/7  LF_LES_1700  "Lift force less than 1700 lbs" %
% Rung: 65 %
SOR LES F8:14 400.0 OTE B3:10/8 EOR
%   F8:14  SCALED_LIFT_FORCE  "Instrument lift strain gage force." %
%   B3:10/8  LF_LES_400  "Lift force less than 400 lbs" %

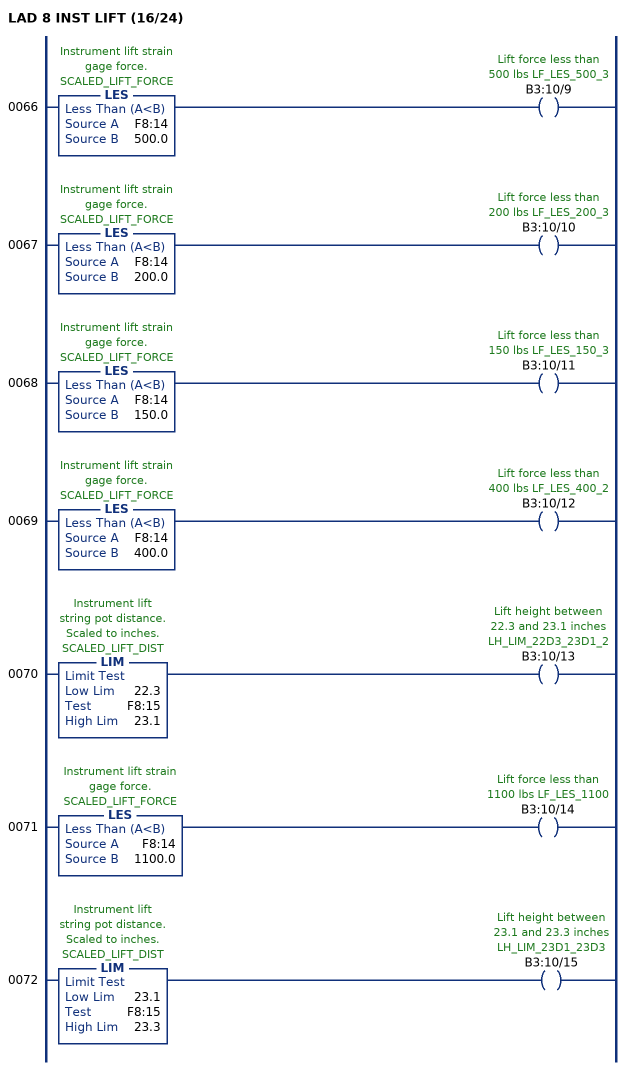
% Rung: 66 %
SOR LES F8:14 500.0 OTE B3:10/9 EOR
%   F8:14  SCALED_LIFT_FORCE  "Instrument lift strain gage force." %
%   B3:10/9  LF_LES_500_3  "Lift force less than 500 lbs" %
% Rung: 67 %
SOR LES F8:14 200.0 OTE B3:10/10 EOR
%   F8:14  SCALED_LIFT_FORCE  "Instrument lift strain gage force." %
%   B3:10/10  LF_LES_200_3  "Lift force less than 200 lbs" %
% Rung: 68 %
SOR LES F8:14 150.0 OTE B3:10/11 EOR
%   F8:14  SCALED_LIFT_FORCE  "Instrument lift strain gage force." %
%   B3:10/11  LF_LES_150_3  "Lift force less than 150 lbs" %
% Rung: 69 %
SOR LES F8:14 400.0 OTE B3:10/12 EOR
%   F8:14  SCALED_LIFT_FORCE  "Instrument lift strain gage force." %
%   B3:10/12  LF_LES_400_2  "Lift force less than 400 lbs" %
% Rung: 70 %
SOR LIM 22.3 F8:15 23.1 OTE B3:10/13 EOR
%   F8:15  SCALED_LIFT_DIST  "Instrument lift string pot distance. Scaled to inches." %
%   B3:10/13  LH_LIM_22D3_23D1_2  "Lift height between 22.3 and 23.1 inches" %
% Rung: 71 %
SOR LES F8:14 1100.0 OTE B3:10/14 EOR
%   F8:14  SCALED_LIFT_FORCE  "Instrument lift strain gage force." %
%   B3:10/14  LF_LES_1100  "Lift force less than 1100 lbs" %
% Rung: 72 %
SOR LIM 23.1 F8:15 23.3 OTE B3:10/15 EOR
%   F8:15  SCALED_LIFT_DIST  "Instrument lift string pot distance. Scaled to inches." %
%   B3:10/15  LH_LIM_23D1_23D3  "Lift height between 23.1 and 23.3 inches" %

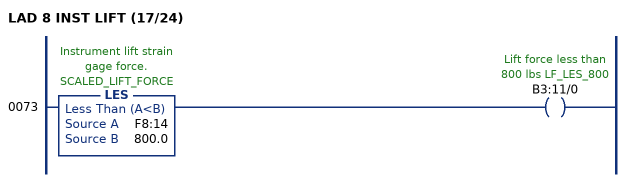
% Rung: 73 %
SOR LES F8:14 800.0 OTE B3:11/0 EOR
%   F8:14  SCALED_LIFT_FORCE  "Instrument lift strain gage force." %
%   B3:11/0  LF_LES_800  "Lift force less than 800 lbs" %

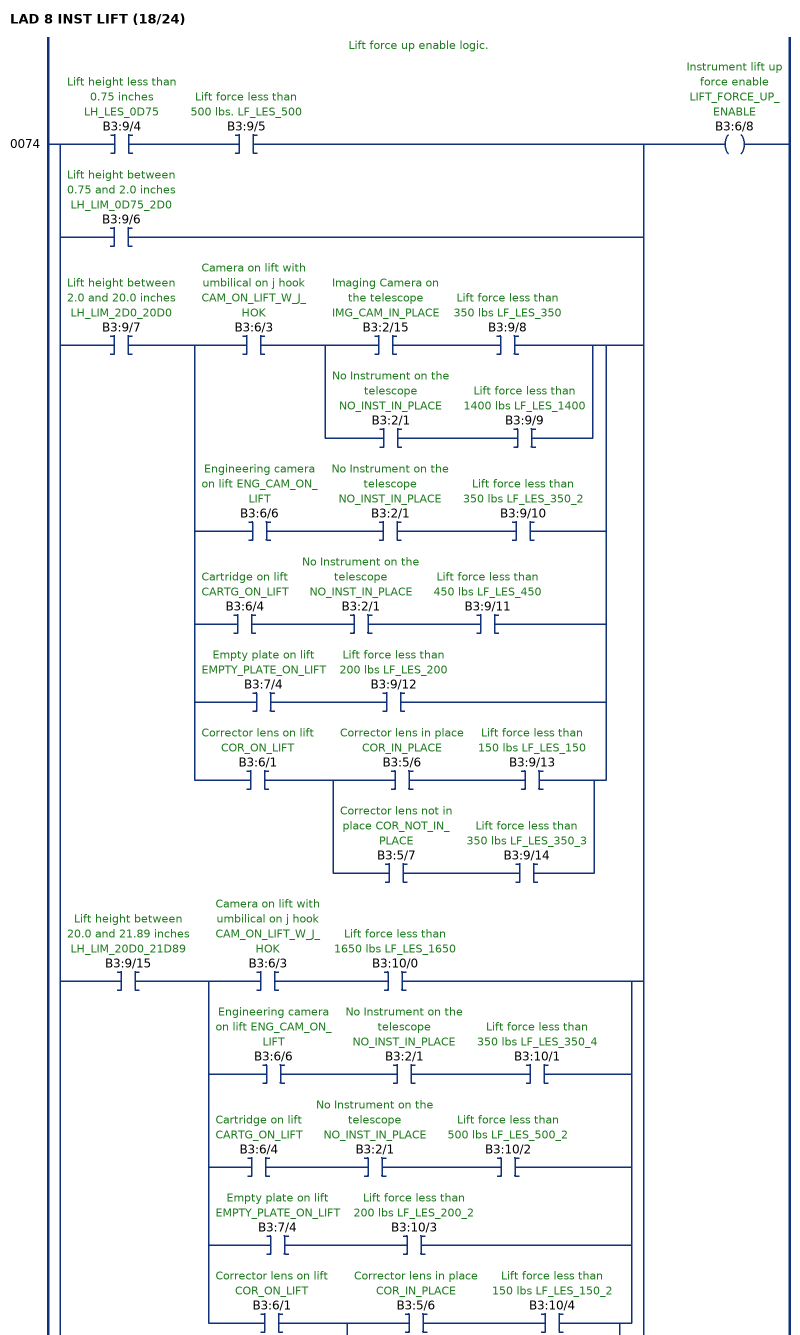

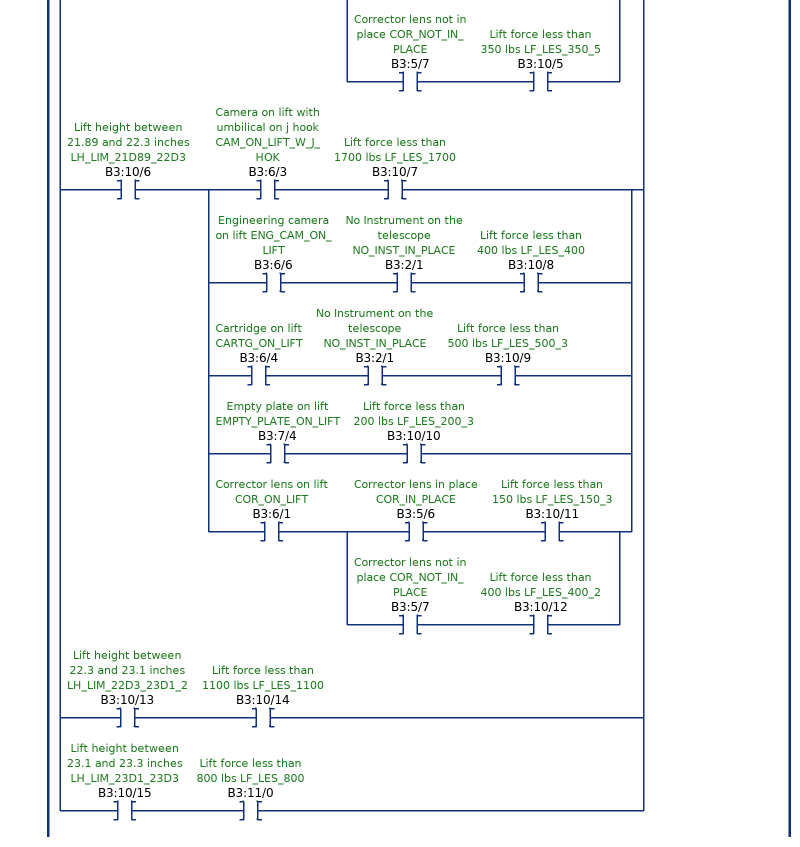
% Rung: 74 %
% Lift force up enable logic. %
SOR BST XIC B3:9/4 XIC B3:9/5 NXB XIC B3:9/6 NXB XIC B3:9/7 BST XIC B3:6/3 BST XIC B3:2/15 XIC B3:9/8 NXB XIC B3:2/1 XIC B3:9/9 BND NXB XIC B3:6/6 XIC B3:2/1 XIC B3:9/10 NXB XIC B3:6/4 XIC B3:2/1 XIC B3:9/11 NXB XIC B3:7/4 XIC B3:9/12 NXB XIC B3:6/1 BST XIC B3:5/6 XIC B3:9/13 NXB XIC B3:5/7 XIC B3:9/14 BND BND NXB XIC B3:9/15 BST XIC B3:6/3 XIC B3:10/0 NXB XIC B3:6/6 XIC B3:2/1 XIC B3:10/1 NXB XIC B3:6/4 XIC B3:2/1 XIC B3:10/2 NXB XIC B3:7/4 XIC B3:10/3 NXB XIC B3:6/1 BST XIC B3:5/6 XIC B3:10/4 NXB XIC B3:5/7 XIC B3:10/5 BND BND NXB XIC B3:10/6 BST XIC B3:6/3 XIC B3:10/7 NXB XIC B3:6/6 XIC B3:2/1 XIC B3:10/8 NXB XIC B3:6/4 XIC B3:2/1 XIC B3:10/9 NXB XIC B3:7/4 XIC B3:10/10 NXB XIC B3:6/1 BST XIC B3:5/6 XIC B3:10/11 NXB XIC B3:5/7 XIC B3:10/12 BND BND NXB XIC B3:10/13 XIC B3:10/14 NXB XIC B3:10/15 XIC B3:11/0 BND OTE B3:6/8 EOR
%   B3:9/4  LH_LES_0D75  "Lift height less than 0.75 inches" %
%   B3:9/5  LF_LES_500  "Lift force less than 500 lbs." %
%   B3:9/6  LH_LIM_0D75_2D0  "Lift height between 0.75 and 2.0 inches" %
%   B3:9/7  LH_LIM_2D0_20D0  "Lift height between 2.0 and 20.0 inches" %
%   B3:6/3  CAM_ON_LIFT_W_J_HOK  "Camera on lift with umbilical on j hook" %
%   B3:2/15  IMG_CAM_IN_PLACE  "Imaging Camera on the telescope" %
%   B3:9/8  LF_LES_350  "Lift force less than 350 lbs" %
%   B3:2/1  NO_INST_IN_PLACE  "No Instrument on the telescope" %
%   B3:9/9  LF_LES_1400  "Lift force less than 1400 lbs" %
%   B3:6/6  ENG_CAM_ON_LIFT  "Engineering camera on lift" %
%   B3:9/10  LF_LES_350_2  "Lift force less than 350 lbs" %
%   B3:6/4  CARTG_ON_LIFT  "Cartridge on lift" %
%   B3:9/11  LF_LES_450  "Lift force less than 450 lbs" %
%   B3:7/4  EMPTY_PLATE_ON_LIFT  "Empty plate on lift" %
%   B3:9/12  LF_LES_200  "Lift force less than 200 lbs" %
%   B3:6/1  COR_ON_LIFT  "Corrector lens on lift" %
%   B3:5/6  COR_IN_PLACE  "Corrector lens in place" %
%   B3:9/13  LF_LES_150  "Lift force less than 150 lbs" %
%   B3:5/7  COR_NOT_IN_PLACE  "Corrector lens not in place" %
%   B3:9/14  LF_LES_350_3  "Lift force less than 350 lbs" %
%   B3:9/15  LH_LIM_20D0_21D89  "Lift height between 20.0 and 21.89 inches" %
%   B3:10/0  LF_LES_1650  "Lift force less than 1650 lbs" %
%   B3:10/1  LF_LES_350_4  "Lift force less than 350 lbs" %
%   B3:10/2  LF_LES_500_2  "Lift force less than 500 lbs" %
%   B3:10/3  LF_LES_200_2  "Lift force less than 200 lbs" %
%   B3:10/4  LF_LES_150_2  "Lift force less than 150 lbs" %
%   B3:10/5  LF_LES_350_5  "Lift force less than 350 lbs" %
%   B3:10/6  LH_LIM_21D89_22D3  "Lift height between 21.89 and 22.3 inches" %
%   B3:10/7  LF_LES_1700  "Lift force less than 1700 lbs" %
%   B3:10/8  LF_LES_400  "Lift force less than 400 lbs" %
%   B3:10/9  LF_LES_500_3  "Lift force less than 500 lbs" %
%   B3:10/10  LF_LES_200_3  "Lift force less than 200 lbs" %
%   B3:10/11  LF_LES_150_3  "Lift force less than 150 lbs" %
%   B3:10/12  LF_LES_400_2  "Lift force less than 400 lbs" %
%   B3:10/13  LH_LIM_22D3_23D1_2  "Lift height between 22.3 and 23.1 inches" %
%   B3:10/14  LF_LES_1100  "Lift force less than 1100 lbs" %
%   B3:10/15  LH_LIM_23D1_23D3  "Lift height between 23.1 and 23.3 inches" %
%   B3:11/0  LF_LES_800  "Lift force less than 800 lbs" %
%   B3:6/8  LIFT_FORCE_UP_ENABLE  "Instrument lift up force enable" %

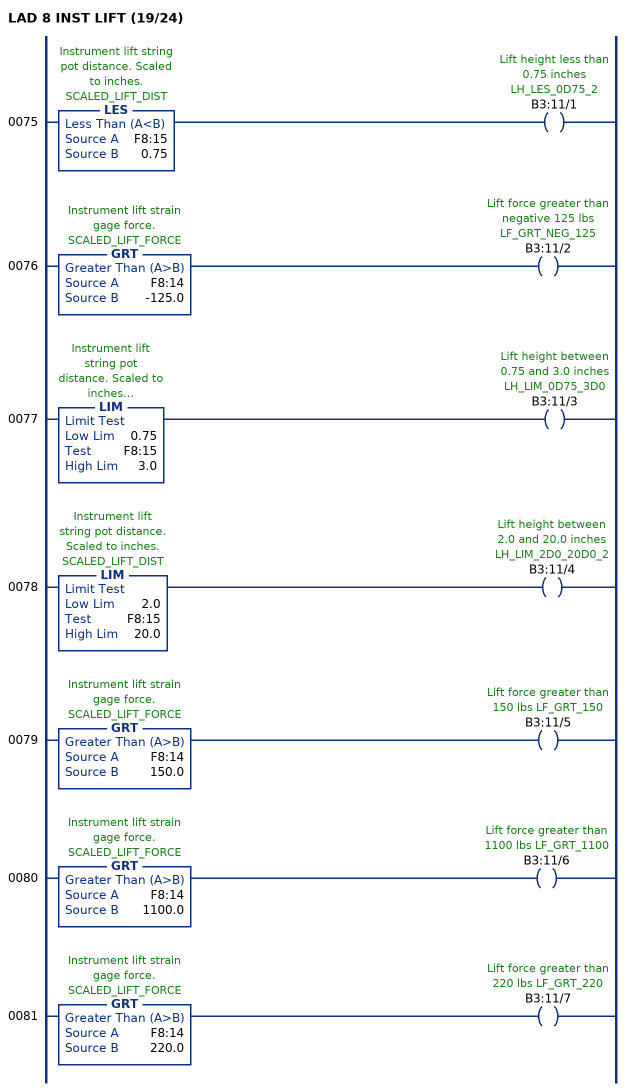
% Rung: 75 %
SOR LES F8:15 0.75 OTE B3:11/1 EOR
%   F8:15  SCALED_LIFT_DIST  "Instrument lift string pot distance. Scaled to inches." %
%   B3:11/1  LH_LES_0D75_2  "Lift height less than 0.75 inches" %
% Rung: 76 %
SOR GRT F8:14 -125.0 OTE B3:11/2 EOR
%   F8:14  SCALED_LIFT_FORCE  "Instrument lift strain gage force." %
%   B3:11/2  LF_GRT_NEG_125  "Lift force greater than negative 125 lbs" %
% Rung: 77 %
SOR LIM 0.75 F8:15 3.0 OTE B3:11/3 EOR
%   F8:15  SCALED_LIFT_DIST  "Instrument lift string pot distance. Scaled to inches." %
%   B3:11/3  LH_LIM_0D75_3D0  "Lift height between 0.75 and 3.0 inches" %
% Rung: 78 %
SOR LIM 2.0 F8:15 20.0 OTE B3:11/4 EOR
%   F8:15  SCALED_LIFT_DIST  "Instrument lift string pot distance. Scaled to inches." %
%   B3:11/4  LH_LIM_2D0_20D0_2  "Lift height between 2.0 and 20.0 inches" %
% Rung: 79 %
SOR GRT F8:14 150.0 OTE B3:11/5 EOR
%   F8:14  SCALED_LIFT_FORCE  "Instrument lift strain gage force." %
%   B3:11/5  LF_GRT_150  "Lift force greater than 150 lbs" %
% Rung: 80 %
SOR GRT F8:14 1100.0 OTE B3:11/6 EOR
%   F8:14  SCALED_LIFT_FORCE  "Instrument lift strain gage force." %
%   B3:11/6  LF_GRT_1100  "Lift force greater than 1100 lbs" %
% Rung: 81 %
SOR GRT F8:14 220.0 OTE B3:11/7 EOR
%   F8:14  SCALED_LIFT_FORCE  "Instrument lift strain gage force." %
%   B3:11/7  LF_GRT_220  "Lift force greater than 220 lbs" %

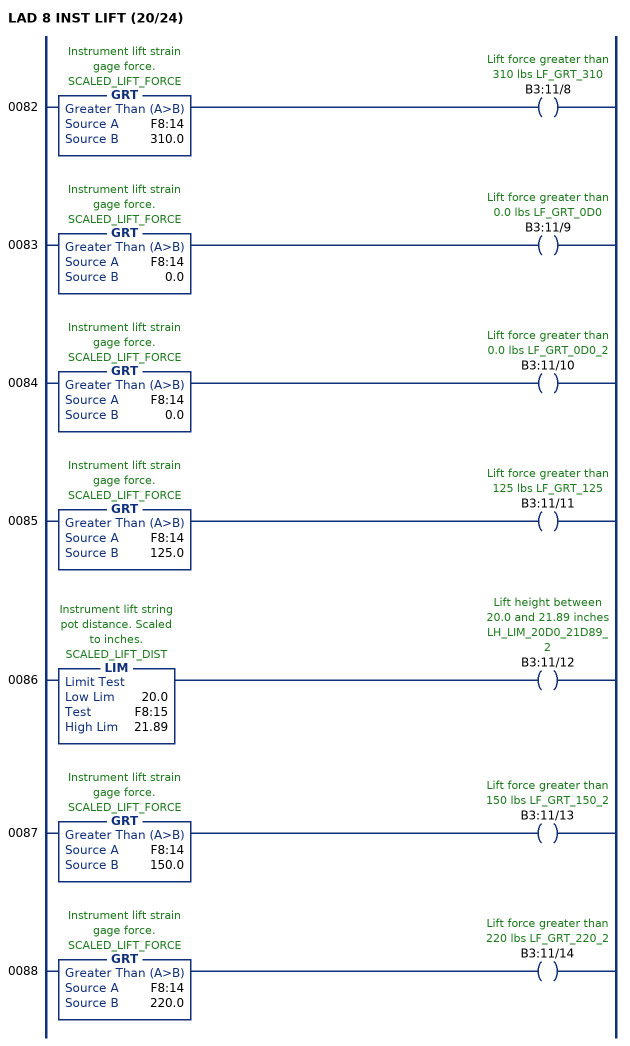
% Rung: 82 %
SOR GRT F8:14 310.0 OTE B3:11/8 EOR
%   F8:14  SCALED_LIFT_FORCE  "Instrument lift strain gage force." %
%   B3:11/8  LF_GRT_310  "Lift force greater than 310 lbs" %
% Rung: 83 %
SOR GRT F8:14 0.0 OTE B3:11/9 EOR
%   F8:14  SCALED_LIFT_FORCE  "Instrument lift strain gage force." %
%   B3:11/9  LF_GRT_0D0  "Lift force greater than 0.0 lbs" %
% Rung: 84 %
SOR GRT F8:14 0.0 OTE B3:11/10 EOR
%   F8:14  SCALED_LIFT_FORCE  "Instrument lift strain gage force." %
%   B3:11/10  LF_GRT_0D0_2  "Lift force greater than 0.0 lbs" %
% Rung: 85 %
SOR GRT F8:14 125.0 OTE B3:11/11 EOR
%   F8:14  SCALED_LIFT_FORCE  "Instrument lift strain gage force." %
%   B3:11/11  LF_GRT_125  "Lift force greater than 125 lbs" %
% Rung: 86 %
SOR LIM 20.0 F8:15 21.89 OTE B3:11/12 EOR
%   F8:15  SCALED_LIFT_DIST  "Instrument lift string pot distance. Scaled to inches." %
%   B3:11/12  LH_LIM_20D0_21D89_2  "Lift height between 20.0 and 21.89 inches" %
% Rung: 87 %
SOR GRT F8:14 150.0 OTE B3:11/13 EOR
%   F8:14  SCALED_LIFT_FORCE  "Instrument lift strain gage force." %
%   B3:11/13  LF_GRT_150_2  "Lift force greater than 150 lbs" %
% Rung: 88 %
SOR GRT F8:14 220.0 OTE B3:11/14 EOR
%   F8:14  SCALED_LIFT_FORCE  "Instrument lift strain gage force." %
%   B3:11/14  LF_GRT_220_2  "Lift force greater than 220 lbs" %

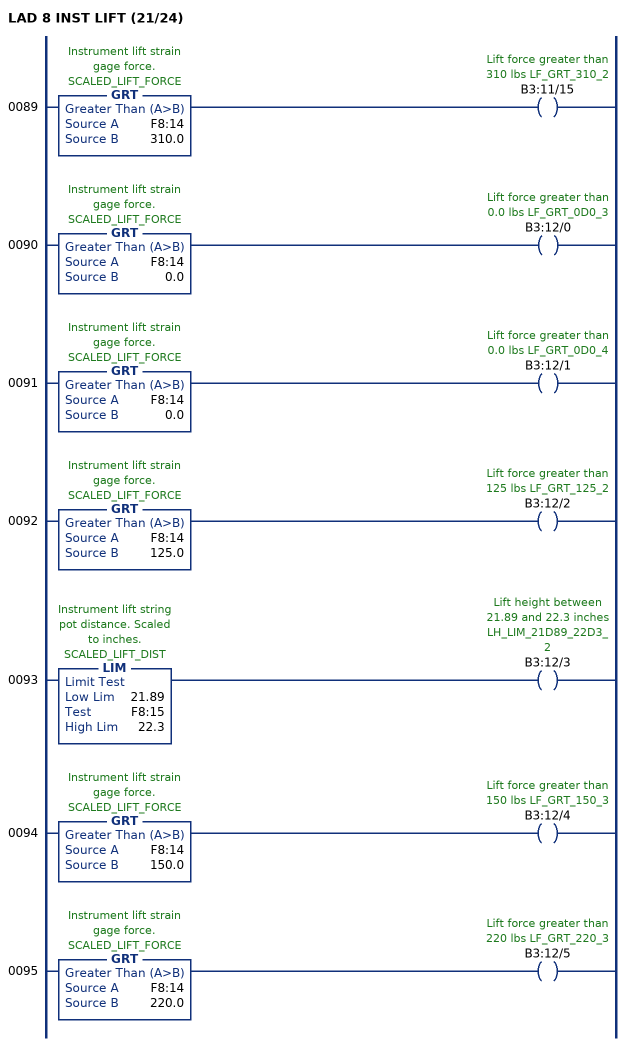
% Rung: 89 %
SOR GRT F8:14 310.0 OTE B3:11/15 EOR
%   F8:14  SCALED_LIFT_FORCE  "Instrument lift strain gage force." %
%   B3:11/15  LF_GRT_310_2  "Lift force greater than 310 lbs" %
% Rung: 90 %
SOR GRT F8:14 0.0 OTE B3:12/0 EOR
%   F8:14  SCALED_LIFT_FORCE  "Instrument lift strain gage force." %
%   B3:12/0  LF_GRT_0D0_3  "Lift force greater than 0.0 lbs" %
% Rung: 91 %
SOR GRT F8:14 0.0 OTE B3:12/1 EOR
%   F8:14  SCALED_LIFT_FORCE  "Instrument lift strain gage force." %
%   B3:12/1  LF_GRT_0D0_4  "Lift force greater than 0.0 lbs" %
% Rung: 92 %
SOR GRT F8:14 125.0 OTE B3:12/2 EOR
%   F8:14  SCALED_LIFT_FORCE  "Instrument lift strain gage force." %
%   B3:12/2  LF_GRT_125_2  "Lift force greater than 125 lbs" %
% Rung: 93 %
SOR LIM 21.89 F8:15 22.3 OTE B3:12/3 EOR
%   F8:15  SCALED_LIFT_DIST  "Instrument lift string pot distance. Scaled to inches." %
%   B3:12/3  LH_LIM_21D89_22D3_2  "Lift height between 21.89 and 22.3 inches" %
% Rung: 94 %
SOR GRT F8:14 150.0 OTE B3:12/4 EOR
%   F8:14  SCALED_LIFT_FORCE  "Instrument lift strain gage force." %
%   B3:12/4  LF_GRT_150_3  "Lift force greater than 150 lbs" %
% Rung: 95 %
SOR GRT F8:14 220.0 OTE B3:12/5 EOR
%   F8:14  SCALED_LIFT_FORCE  "Instrument lift strain gage force." %
%   B3:12/5  LF_GRT_220_3  "Lift force greater than 220 lbs" %

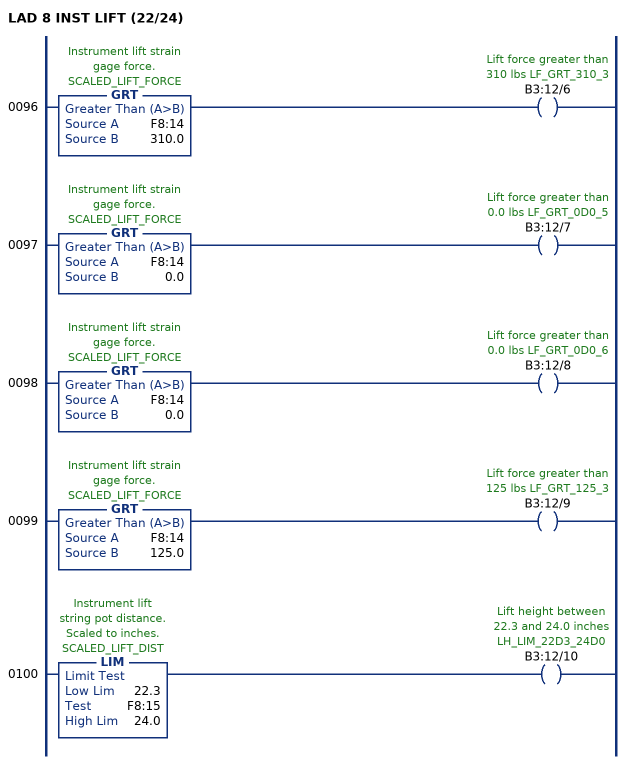
% Rung: 96 %
SOR GRT F8:14 310.0 OTE B3:12/6 EOR
%   F8:14  SCALED_LIFT_FORCE  "Instrument lift strain gage force." %
%   B3:12/6  LF_GRT_310_3  "Lift force greater than 310 lbs" %
% Rung: 97 %
SOR GRT F8:14 0.0 OTE B3:12/7 EOR
%   F8:14  SCALED_LIFT_FORCE  "Instrument lift strain gage force." %
%   B3:12/7  LF_GRT_0D0_5  "Lift force greater than 0.0 lbs" %
% Rung: 98 %
SOR GRT F8:14 0.0 OTE B3:12/8 EOR
%   F8:14  SCALED_LIFT_FORCE  "Instrument lift strain gage force." %
%   B3:12/8  LF_GRT_0D0_6  "Lift force greater than 0.0 lbs" %
% Rung: 99 %
SOR GRT F8:14 125.0 OTE B3:12/9 EOR
%   F8:14  SCALED_LIFT_FORCE  "Instrument lift strain gage force." %
%   B3:12/9  LF_GRT_125_3  "Lift force greater than 125 lbs" %
% Rung: 100 %
SOR LIM 22.3 F8:15 24.0 OTE B3:12/10 EOR
%   F8:15  SCALED_LIFT_DIST  "Instrument lift string pot distance. Scaled to inches." %
%   B3:12/10  LH_LIM_22D3_24D0  "Lift height between 22.3 and 24.0 inches" %

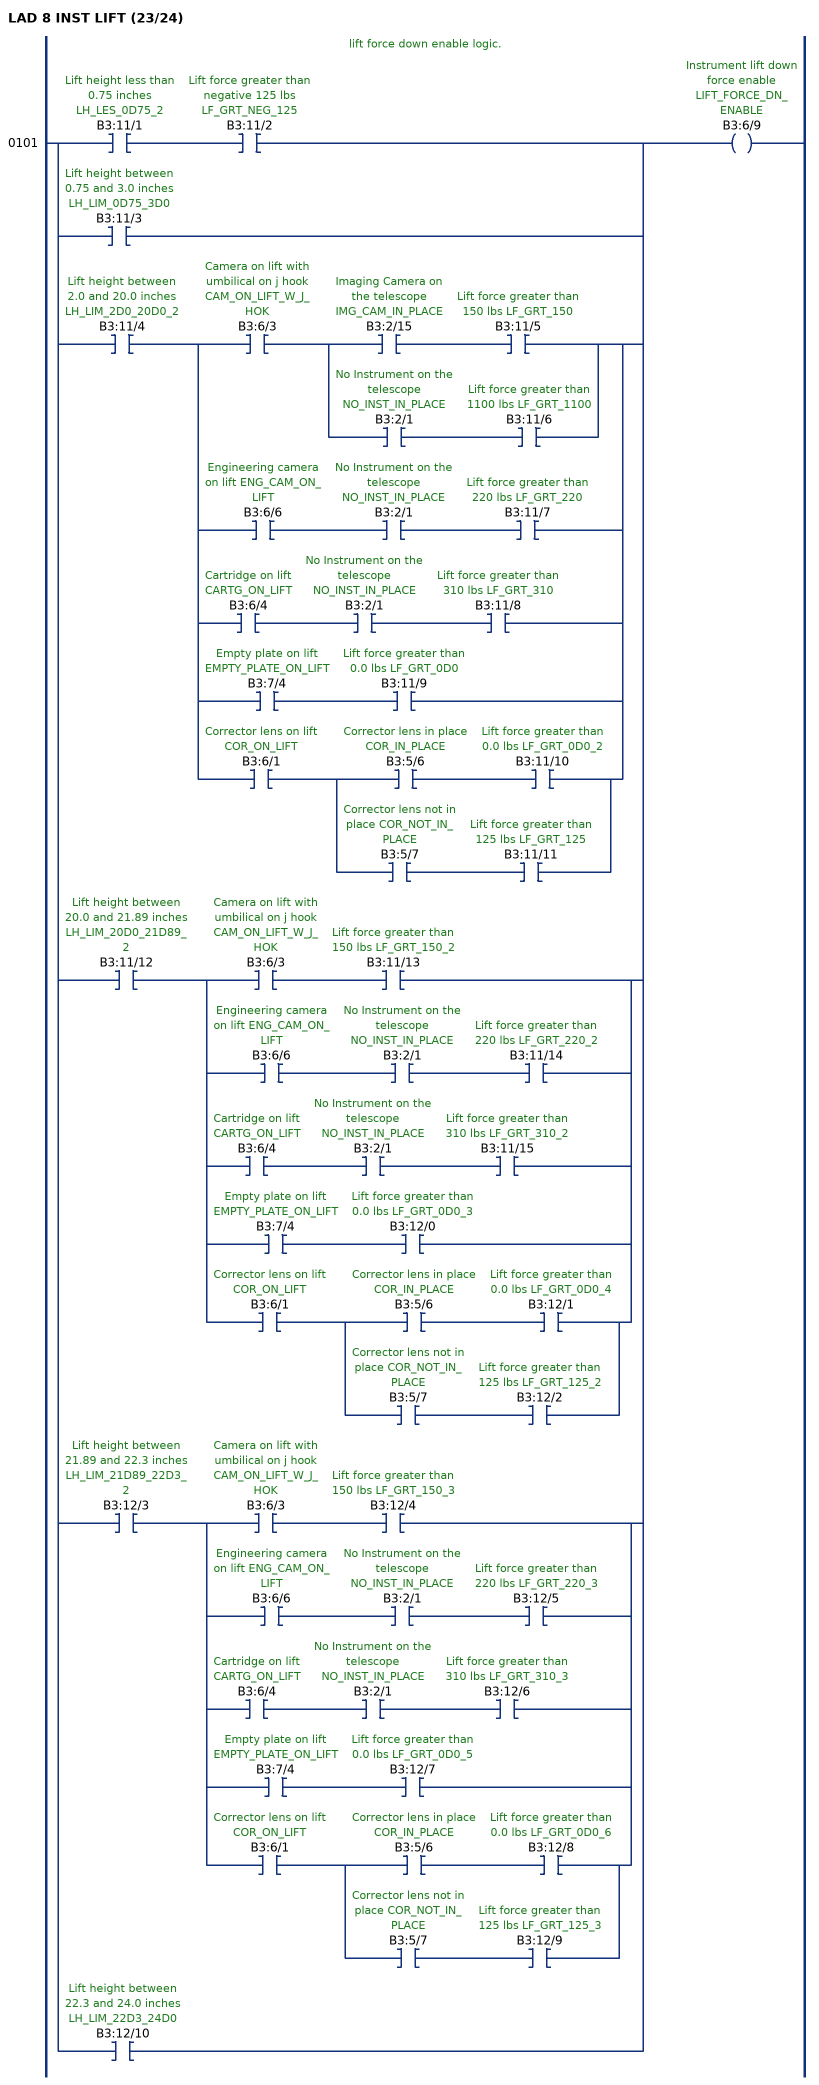
% Rung: 101 %
% lift force down enable logic. %
SOR BST XIC B3:11/1 XIC B3:11/2 NXB XIC B3:11/3 NXB XIC B3:11/4 BST XIC B3:6/3 BST XIC B3:2/15 XIC B3:11/5 NXB XIC B3:2/1 XIC B3:11/6 BND NXB XIC B3:6/6 XIC B3:2/1 XIC B3:11/7 NXB XIC B3:6/4 XIC B3:2/1 XIC B3:11/8 NXB XIC B3:7/4 XIC B3:11/9 NXB XIC B3:6/1 BST XIC B3:5/6 XIC B3:11/10 NXB XIC B3:5/7 XIC B3:11/11 BND BND NXB XIC B3:11/12 BST XIC B3:6/3 XIC B3:11/13 NXB XIC B3:6/6 XIC B3:2/1 XIC B3:11/14 NXB XIC B3:6/4 XIC B3:2/1 XIC B3:11/15 NXB XIC B3:7/4 XIC B3:12/0 NXB XIC B3:6/1 BST XIC B3:5/6 XIC B3:12/1 NXB XIC B3:5/7 XIC B3:12/2 BND BND NXB XIC B3:12/3 BST XIC B3:6/3 XIC B3:12/4 NXB XIC B3:6/6 XIC B3:2/1 XIC B3:12/5 NXB XIC B3:6/4 XIC B3:2/1 XIC B3:12/6 NXB XIC B3:7/4 XIC B3:12/7 NXB XIC B3:6/1 BST XIC B3:5/6 XIC B3:12/8 NXB XIC B3:5/7 XIC B3:12/9 BND BND NXB XIC B3:12/10 BND OTE B3:6/9 EOR
%   B3:11/1  LH_LES_0D75_2  "Lift height less than 0.75 inches" %
%   B3:11/2  LF_GRT_NEG_125  "Lift force greater than negative 125 lbs" %
%   B3:11/3  LH_LIM_0D75_3D0  "Lift height between 0.75 and 3.0 inches" %
%   B3:11/4  LH_LIM_2D0_20D0_2  "Lift height between 2.0 and 20.0 inches" %
%   B3:6/3  CAM_ON_LIFT_W_J_HOK  "Camera on lift with umbilical on j hook" %
%   B3:2/15  IMG_CAM_IN_PLACE  "Imaging Camera on the telescope" %
%   B3:11/5  LF_GRT_150  "Lift force greater than 150 lbs" %
%   B3:2/1  NO_INST_IN_PLACE  "No Instrument on the telescope" %
%   B3:11/6  LF_GRT_1100  "Lift force greater than 1100 lbs" %
%   B3:6/6  ENG_CAM_ON_LIFT  "Engineering camera on lift" %
%   B3:11/7  LF_GRT_220  "Lift force greater than 220 lbs" %
%   B3:6/4  CARTG_ON_LIFT  "Cartridge on lift" %
%   B3:11/8  LF_GRT_310  "Lift force greater than 310 lbs" %
%   B3:7/4  EMPTY_PLATE_ON_LIFT  "Empty plate on lift" %
%   B3:11/9  LF_GRT_0D0  "Lift force greater than 0.0 lbs" %
%   B3:6/1  COR_ON_LIFT  "Corrector lens on lift" %
%   B3:5/6  COR_IN_PLACE  "Corrector lens in place" %
%   B3:11/10  LF_GRT_0D0_2  "Lift force greater than 0.0 lbs" %
%   B3:5/7  COR_NOT_IN_PLACE  "Corrector lens not in place" %
%   B3:11/11  LF_GRT_125  "Lift force greater than 125 lbs" %
%   B3:11/12  LH_LIM_20D0_21D89_2  "Lift height between 20.0 and 21.89 inches" %
%   B3:11/13  LF_GRT_150_2  "Lift force greater than 150 lbs" %
%   B3:11/14  LF_GRT_220_2  "Lift force greater than 220 lbs" %
%   B3:11/15  LF_GRT_310_2  "Lift force greater than 310 lbs" %
%   B3:12/0  LF_GRT_0D0_3  "Lift force greater than 0.0 lbs" %
%   B3:12/1  LF_GRT_0D0_4  "Lift force greater than 0.0 lbs" %
%   B3:12/2  LF_GRT_125_2  "Lift force greater than 125 lbs" %
%   B3:12/3  LH_LIM_21D89_22D3_2  "Lift height between 21.89 and 22.3 inches" %
%   B3:12/4  LF_GRT_150_3  "Lift force greater than 150 lbs" %
%   B3:12/5  LF_GRT_220_3  "Lift force greater than 220 lbs" %
%   B3:12/6  LF_GRT_310_3  "Lift force greater than 310 lbs" %
%   B3:12/7  LF_GRT_0D0_5  "Lift force greater than 0.0 lbs" %
%   B3:12/8  LF_GRT_0D0_6  "Lift force greater than 0.0 lbs" %
%   B3:12/9  LF_GRT_125_3  "Lift force greater than 125 lbs" %
%   B3:12/10  LH_LIM_22D3_24D0  "Lift height between 22.3 and 24.0 inches" %
%   B3:6/9  LIFT_FORCE_DN_ENABLE  "Instrument lift down force enable" %

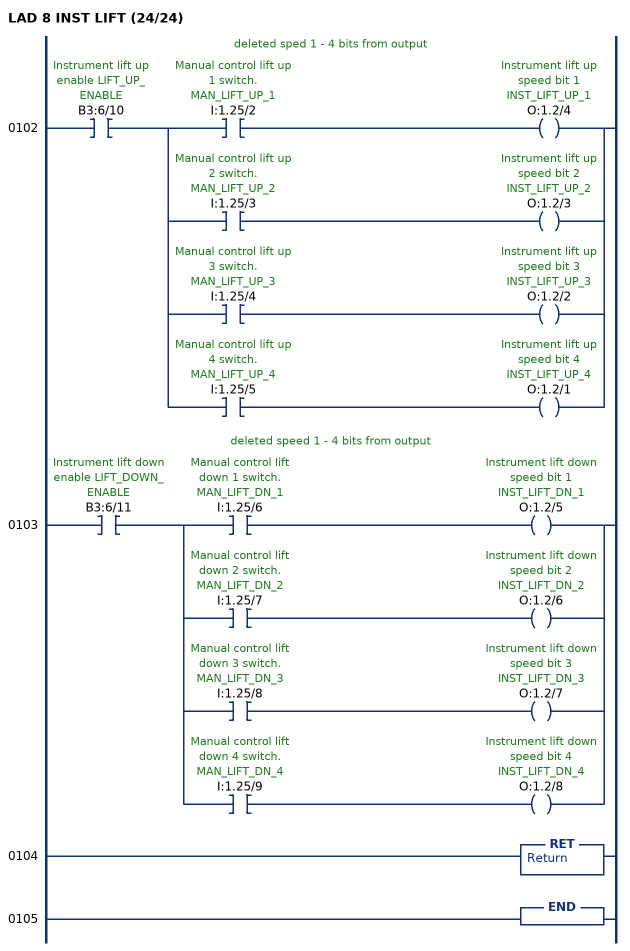
% Rung: 102 %
% deleted sped 1 - 4 bits from output %
SOR XIC B3:6/10 BST XIC I:1.25/2 OTE O:1.2/4 NXB XIC I:1.25/3 OTE O:1.2/3 NXB XIC I:1.25/4 OTE O:1.2/2 NXB XIC I:1.25/5 OTE O:1.2/1 BND EOR
%   B3:6/10  LIFT_UP_ENABLE  "Instrument lift up enable" %
%   I:1.25/2  MAN_LIFT_UP_1  "Manual control lift up 1 switch." %
%   O:1.2/4  INST_LIFT_UP_1  "Instrument lift up speed bit 1" %
%   I:1.25/3  MAN_LIFT_UP_2  "Manual control lift up 2 switch." %
%   O:1.2/3  INST_LIFT_UP_2  "Instrument lift up speed bit 2" %
%   I:1.25/4  MAN_LIFT_UP_3  "Manual control lift up 3 switch." %
%   O:1.2/2  INST_LIFT_UP_3  "Instrument lift up speed bit 3" %
%   I:1.25/5  MAN_LIFT_UP_4  "Manual control lift up 4 switch." %
%   O:1.2/1  INST_LIFT_UP_4  "Instrument lift up speed bit 4" %
% Rung: 103 %
% deleted speed 1 - 4 bits from output %
SOR XIC B3:6/11 BST XIC I:1.25/6 OTE O:1.2/5 NXB XIC I:1.25/7 OTE O:1.2/6 NXB XIC I:1.25/8 OTE O:1.2/7 NXB XIC I:1.25/9 OTE O:1.2/8 BND EOR
%   B3:6/11  LIFT_DOWN_ENABLE  "Instrument lift down enable" %
%   I:1.25/6  MAN_LIFT_DN_1  "Manual control lift down 1 switch." %
%   O:1.2/5  INST_LIFT_DN_1  "Instrument lift down speed bit 1" %
%   I:1.25/7  MAN_LIFT_DN_2  "Manual control lift down 2 switch." %
%   O:1.2/6  INST_LIFT_DN_2  "Instrument lift down speed bit 2" %
%   I:1.25/8  MAN_LIFT_DN_3  "Manual control lift down 3 switch." %
%   O:1.2/7  INST_LIFT_DN_3  "Instrument lift down speed bit 3" %
%   I:1.25/9  MAN_LIFT_DN_4  "Manual control lift down 4 switch." %
%   O:1.2/8  INST_LIFT_DN_4  "Instrument lift down speed bit 4" %
% Rung: 104 %
SOR RET EOR
% Rung: 105 %
SOR END EOR

LADDER 9 "INST LATCH"    % Instrument Latch Control Box File %
